		// Remove empty index in buffer by moving next alarms.
		// IF positions in buffer are not empty (trigger false)
		diWarningLoop := diBufferIdToRemove;
		
		WHILE diWarningLoop < HEVS_PackTag_GVL.C_ADMIN_MAXWARNINGS AND 
              stAdminWarning[diWarningLoop + 1].Trigger       DO
			// Cannot be out of buffer because diAlarmLoop < GVL_PackConstant.ALARM_EXTENT
			// Move buffer (n+1) to buffer(n)
			stAdminWarning[diWarningLoop] := stAdminWarning[diWarningLoop + 1]; 
			diWarningLoop := diWarningLoop + 1;
		END_WHILE
		
		// Erase last position on buffer.
		IF diWarningLoop <> diBufferIdToRemove THEN
			stAdminWarning[diWarningLoop].AckDateTime := DT#1970-1-1-0:0:0;
			stAdminWarning[diWarningLoop].Category := 0;
			stAdminWarning[diWarningLoop].DateTime := DT#1970-1-1-0:0:0;
			stAdminWarning[diWarningLoop].ID := 0;
			stAdminWarning[diWarningLoop].Message := '';
			stAdminWarning[diWarningLoop].Trigger := FALSE;
			stAdminWarning[diWarningLoop].Value := 0;
		END_IF
	END_IF 
END_IF

(*
	Set AckDateTime
	Do not set if NOT bSetAlarm because Event was removed with the above code.
	
	Acknowledge on rising edge only
*)
rTrigAck(CLK := bAckWarningTrig);

IF rTrigAck.Q AND bSetWarning THEN
	FOR diWarningLoop := 0 TO HEVS_PackTag_GVL.C_ADMIN_MAXWARNINGS BY 1 DO
		IF (stAdminWarning[diWarningLoop].ID = ID) THEN
			stAdminWarning[diWarningLoop].AckDateTime := PackTag.Admin.PLCDateTime;
		END_IF
	END_FOR	
END_IF


                
END_FUNCTION_BLOCK

(* A function block to set an alarm using PackML 2022 structure TwinCAT Tc3_EventLogger Source: www.hevs.ch Author: Cedric Lenoir Date: 22 August 2024 *)
FUNCTION_BLOCK FB_HEVS_StopReason
  VAR_INPUT
    SuspendCategory : DINT := 1;  (* With default value 1 *)
    HoldCategory : DINT := 2;  (* With default value 2 *)
    StopCategory : DINT := 3;  (* With default value 3 *)
    AbortCategory : DINT := 4;  (* With default value 4 *)
    CompleteCategory : DINT := 6;  (* With default value 6 *)
  END_VAR
  VAR_IN_OUT
    stStopReason : HEVS_PackTag_Event;
    stAdminAlarm : ARRAY[0..HEVS_PackTag_GVL.C_ADMIN_MAXALARMS] OF HEVS_PackTag_Event;
  END_VAR
  VAR_OUTPUT
    SuspendCmd : BOOL;
    HoldCmd : BOOL;
    StopCmd : BOOL;
    AbortCmd : BOOL;
    CompleteCmd : BOOL;
    stopReasonToMaster : E_PackCmd := E_PackCmd.eUndefined;  (* Use to activate Stop Reason on FB_PackMasterState *)
  END_VAR
  VAR
    SuspendExistInAlarm : BOOL;
    HoldExistInAlarm : BOOL;
    StopExistInAlarm : BOOL;
    AbortExistInAlarm : BOOL;
    CompleteExistInAlarm : BOOL;
    SuspendId : DINT;
    HoldId : DINT;
    StopId : DINT;
    AbortId : DINT;
    CompleteId : DINT;
    diAlarmLoop : DINT;
  END_VAR

                  (*
	TR 88 not precise, 
	we will show the Cmd with the Highest Priority
	with Abort, the higest, Stop, Complete, Hold and Suspend, the lowest.
*)
SuspendExistInAlarm := FALSE;
HoldExistInAlarm := FALSE;
StopExistInAlarm := FALSE;
AbortExistInAlarm := FALSE;
CompleteExistInAlarm := FALSE;

SuspendId := 0;
HoldId := 0;
StopId := 0;
AbortId := 0;
CompleteId := 0;
	
FOR diAlarmLoop := 0 TO HEVS_PackTag_GVL.C_ADMIN_MAXALARMS BY 1 DO
	IF stAdminAlarm[diAlarmLoop].Category = SuspendCategory THEN
		SuspendExistInAlarm := TRUE;
		SuspendId := diAlarmLoop;
	END_IF

	IF stAdminAlarm[diAlarmLoop].Category = HoldCategory THEN
		HoldExistInAlarm := TRUE;
		HoldId := diAlarmLoop;
	END_IF

	IF stAdminAlarm[diAlarmLoop].Category = StopCategory THEN
		StopExistInAlarm := TRUE;
		StopId := diAlarmLoop;
	END_IF

	IF stAdminAlarm[diAlarmLoop].Category = AbortCategory THEN
		AbortExistInAlarm := TRUE;
		AbortId := diAlarmLoop;
	END_IF

	IF stAdminAlarm[diAlarmLoop].Category = CompleteCategory THEN
		CompleteExistInAlarm := TRUE;
		CompleteId := diAlarmLoop;
	END_IF
END_FOR

// Select the highest priority sto reason
IF AbortExistInAlarm THEN
	stStopReason := stAdminAlarm[AbortId];
	stopReasonToMaster := E_PackCmd.eAbort;
	
ELSIF StopExistInAlarm THEN
	stStopReason := stAdminAlarm[StopId];
	stopReasonToMaster := E_PackCmd.eStop;

ELSIF CompleteExistInAlarm THEN
	stStopReason := stAdminAlarm[CompleteId];
	stopReasonToMaster := E_PackCmd.eComplete;
	
ELSIF HoldExistInAlarm THEN
	stStopReason := stAdminAlarm[HoldId];
	stopReasonToMaster := E_PackCmd.eHold;
	
ELSIF SuspendExistInAlarm THEN
	stStopReason := stAdminAlarm[SuspendId];
	stopReasonToMaster := E_PackCmd.eSuspend;
	
ELSE // No Stop reason, reset
	stStopReason.AckDateTime := DT#1970-1-1-0:0:0;
	stStopReason.Category := 0;
	stStopReason.DateTime := DT#1970-1-1-0:0:0;
	stStopReason.ID := 0;
	stStopReason.Message := '';
	stStopReason.Trigger := FALSE;
	stStopReason.Value := 0; 

	stopReasonToMaster := E_PackCmd.eUndefined;
END_IF

(*
	Set outputs
*)
AbortCmd := AbortExistInAlarm;
StopCmd := StopExistInAlarm AND NOT AbortExistInAlarm;
CompleteCmd := CompleteExistInAlarm AND NOT (AbortExistInAlarm OR StopExistInAlarm);
HoldCmd := HoldExistInAlarm AND NOT (AbortExistInAlarm OR StopExistInAlarm OR CompleteExistInAlarm);
SuspendCmd := SuspendCmd AND NOT (AbortExistInAlarm OR StopExistInAlarm OR CompleteExistInAlarm OR HoldExistInAlarm);



                
END_FUNCTION_BLOCK

(* A function block of type Enable Source: www.hevs.ch Author: Cedric Lenoir Date: 22 August 2024 *)
FUNCTION_BLOCK FB_InOpBase
  VAR_INPUT
    Enable : BOOL;
  END_VAR
  VAR_OUTPUT
    InOperation : BOOL;
    Error : BOOL;
    ErrorId : WORD;
  END_VAR
  VAR
    eOperationBase : E_InOperationBase;
    errorCondition : BOOL;
  END_VAR

                  // Read Input

CASE eOperationBase OF
	E_InOperationBase.Idle 			:
		IF Enable THEN
			eOperationBase := E_InOperationBase.Init;
		END_IF
        
	E_InOperationBase.Init 			:
		IF NOT Enable THEN
			eOperationBase := E_InOperationBase.Idle;
		ELSIF errorCondition THEN
			eOperationBase := E_InOperationBase.Error;
		END_IF
        
	E_InOperationBase.InOp  :
		IF NOT Enable THEN
			eOperationBase := E_InOperationBase.Idle;
		ELSIF errorCondition THEN
			eOperationBase := E_InOperationBase.Error;
		END_IF
        
	E_InOperationBase.Error			:
		IF NOT Enable THEN
			eOperationBase := E_InOperationBase.Idle;
		END_IF
END_CASE

InOperation := eOperationBase = E_InOperationBase.InOp;
			   
Error := (eOperationBase = E_InOperationBase.Error);

// 0 while no ID defined
ErrorId := 0;
                
END_FUNCTION_BLOCK

PROGRAM PRG_Sandbox
  VAR
    uliLoop : ULINT;
    bInit : BOOL;  (* Only used to give a basic value to some variables. *)
    fbInOpBase : FB_InOpBase;
    fbExecuteDone : FB_ExecuteDone;
  END_VAR

                  (*
    Test base FB
*)
fbInOpBase();
fbExecuteDone();

uliLoop := uliLoop + 1;
(*
    Used to test connection with Node-RED via ADS
*)
ACT_TestNode();


                

ACTION ACT_TestNode:
                      (*
    This part is only used to test the communication with Node-RED
*)
IF NOT bInit THEN
    bInit := TRUE;
    GVL_Node.readREAL    := 3.14;
    GVL_Node.readDINT    := 421;
    GVL_Node.readBOOL    := TRUE;
    GVL_Node.readString  := 'Empty';
    GVL_Node.writeREAL   := 0;
    GVL_Node.writeDINT   := 0;
    GVL_Node.writeBOOL   := FALSE;
END_IF

IF GVL_Node.readREAL > 6.28 THEN
    GVL_Node.readREAL := 0;
ELSE
    GVL_Node.readREAL := GVL_Node.readREAL + 0.1; ;
END_IF
    
IF GVL_Node.readDINT > 1000 THEN
    GVL_Node.readDINT := 0;
ELSE
    GVL_Node.readDINT := GVL_Node.readDINT + 1;
END_IF
                    
END_ACTION
END_PROGRAM

(* www.hevs.ch Institut Systemes Industriels Project: HEVS Pack 2022 Author: Cedric Lenoir Date: 2024 August 29 This program is done to test alarms with a set of 3 Alarms 3 Warnings *)
PROGRAM PRG_TestAlarm
  VAR
    BuildUiString : STRING;  (* Tempo var to display an evant in String Format for UI *)
    fbSetAlarm_0 : FB_HEVS_SetAlarm;  (* Test alarms with FB first *)
    fbSetAlarm_1 : FB_HEVS_SetAlarm;
    fbSetAlarm_2 : FB_HEVS_SetAlarm;
    fbSetWarning_0 : FB_HEVS_SetWarning;
    fbSetWarning_1 : FB_HEVS_SetWarning;
    fbSetWarning_2 : FB_HEVS_SetWarning;
  END_VAR

                  (*
	Call some alarms for test
*) 
fbSetAlarm_0(// Bit activation of Alarm and Ack
			 bSetAlarm := PackTag.hevsPackAlarm_UI.uiSetAlarm_0,
	         bAckAlarmTrig := PackTag.hevsPackAlarm_UI.uiAckAlarm_0,
			 // Alarm Parameters
			 ID := 5,
	         Value := 35,
	         Message := 'Abort 4, E-Stop',
	         Category := E_EventCategory.Abort,
			 // Reference to plc time from PackTag
			 plcDateTimePack	:= PackTag.Admin.PLCDateTime,
			 // Link to PackTag Admin
	         stAdminAlarm := PackTag.Admin.Alarm,
			 stAdminAlarmHistory := PackTag.Admin.AlarmHistory);
			 
fbSetAlarm_1(bSetAlarm := PackTag.hevsPackAlarm_UI.uiSetAlarm_1,
	         bAckAlarmTrig := PackTag.hevsPackAlarm_UI.uiAckAlarm_1,
			 ID := 6,
	         Value := 36,
	         Message := 'Stop 3, Motor Hot',
	         Category := E_EventCategory.Stop,
			 // Reference to plc time from PackTag
			 plcDateTimePack	:= PackTag.Admin.PLCDateTime,
			 // Link to PackTag Admin
	         stAdminAlarm := PackTag.Admin.Alarm,
			 stAdminAlarmHistory := PackTag.Admin.AlarmHistory);


fbSetAlarm_2(bSetAlarm := PackTag.hevsPackAlarm_UI.uiSetAlarm_2,
	         bAckAlarmTrig := PackTag.hevsPackAlarm_UI.uiAckAlarm_2,
			 ID := 7,
	         Value := 37,
	         Message := 'Hold 2, Gripper not closed',
	         Category := E_EventCategory.Hold,
			 // Reference to plc time from PackTag
			 plcDateTimePack	:= PackTag.Admin.PLCDateTime,
			 // Link to PackTag Admin
	         stAdminAlarm := PackTag.Admin.Alarm,
			 stAdminAlarmHistory := PackTag.Admin.AlarmHistory);	

(*
	Call some warnings for test
*)
fbSetWarning_0(bSetWarning := PackTag.hevsPackAlarm_UI.uiSetWarning_0,
	           bAckWarningTrig := PackTag.hevsPackAlarm_UI.uiAckWarning_0,
			   // Warning Parameters
			   ID := 1,
	           Value := 31,
	           Message := 'Warning 0, Door Open',
	           Category := E_EventCategory.Warning,
			   // Reference to plc time from PackTag
			   plcDateTimePack	:= PackTag.Admin.PLCDateTime,
			   // Link to PackTag Admin
	           stAdminWarning := PackTag.Admin.Warning);
			 
fbSetWarning_1(bSetWarning := PackTag.hevsPackAlarm_UI.uiSetWarning_1,
	           bAckWarningTrig := PackTag.hevsPackAlarm_UI.uiAckWarning_1,
			   // Warning Parameters
			   ID := 2,
	           Value := 32,
	           Message := 'Warning 1, Loaded',
	           Category := E_EventCategory.Warning,
			   // Reference to plc time from PackTag
			   plcDateTimePack	:= PackTag.Admin.PLCDateTime,
			   // Link to PackTag Admin
	           stAdminWarning := PackTag.Admin.Warning);


fbSetWarning_2(bSetWarning := PackTag.hevsPackAlarm_UI.uiSetWarning_2,
	           bAckWarningTrig := PackTag.hevsPackAlarm_UI.uiAckWarning_2,
			   // Warning Parameters
			   ID := 3,
	           Value := 33,
	           Message := 'Warning 3, Finished',
	           Category := E_EventCategory.Warning,
			   // Reference to plc time from PackTag
			   plcDateTimePack	:= PackTag.Admin.PLCDateTime,
			   // Link to PackTag Admin
	           stAdminWarning := PackTag.Admin.Warning);						 

// Display first evant in UI in string format.
// Could add History too.
ACT_Build_Ui_Strings();


			 		 

                

ACTION ACT_Build_Ui_Strings:
                      (*
	Send to UI:	First line of Alarms
				First line of Warning
				Stop reason
*)
//PackTag.hevsPackAlarm_UI.uiTextAlarmOne := 'Complete with first Alarm';
BuildUiString := DINT_TO_STRING(PackTag.Admin.Alarm[0].ID);
BuildUiString := CONCAT(BuildUiString, ' ');
BuildUiString := CONCAT(BuildUiString, PackTag.Admin.Alarm[0].Message);
BuildUiString := CONCAT(BuildUiString, ' ');
BuildUiString := CONCAT(BuildUiString, DINT_TO_STRING(PackTag.Admin.Alarm[0].Category));
BuildUiString := CONCAT(BuildUiString, ' ');
BuildUiString := CONCAT(BuildUiString, DT_TO_STRING(PackTag.Admin.Alarm[0].DateTime));
PackTag.hevsPackAlarm_UI.uiTextAlarmOne := BuildUiString; 


BuildUiString := DINT_TO_STRING(PackTag.Admin.Warning[0].ID);
BuildUiString := CONCAT(BuildUiString, ' ');
BuildUiString := CONCAT(BuildUiString, PackTag.Admin.Warning[0].Message);
BuildUiString := CONCAT(BuildUiString, ' ');
BuildUiString := CONCAT(BuildUiString, DINT_TO_STRING(PackTag.Admin.Warning[0].Category));
BuildUiString := CONCAT(BuildUiString, ' ');
BuildUiString := CONCAT(BuildUiString, DT_TO_STRING(PackTag.Admin.Warning[0].DateTime));
PackTag.hevsPackAlarm_UI.uiTextWarningOne := BuildUiString;

BuildUiString := DINT_TO_STRING(PackTag.Admin.StopReason.ID);
BuildUiString := CONCAT(BuildUiString, ' ');
BuildUiString := CONCAT(BuildUiString, PackTag.Admin.StopReason.Message);
BuildUiString := CONCAT(BuildUiString, ' ');
BuildUiString := CONCAT(BuildUiString, DINT_TO_STRING(PackTag.Admin.StopReason.Category));
BuildUiString := CONCAT(BuildUiString, ' ');
BuildUiString := CONCAT(BuildUiString, DT_TO_STRING(PackTag.Admin.StopReason.DateTime));
PackTag.hevsPackAlarm_UI.uiTextStopReason := BuildUiString;


                    
END_ACTION
END_PROGRAM

(* www.hevs.ch Institut Systemes Industriels Project: HEVS Pack 2022 Author: Cedric Lenoir Date: 2024 August 30 This Function Block compute time statistics *)
FUNCTION_BLOCK FB_PackStatistic
  VAR_INPUT
    Enable : BOOL;
  END_VAR
  VAR_IN_OUT
    plcCurrentTime_s : UDINT;  (* E.g from PackTag.hevsPackTime.Local_date_time_seconds *)
    unitCurrentMode : E_PackModes;
    unitCurrentState : E_PackState;
    unitAdmin : HEVS_PackTag_Admin;
  END_VAR
  VAR_OUTPUT
    Active : BOOL;
  END_VAR
  VAR
    trigModeTimeCurrent : R_TRIG;  (* Detext State / Mode change *)
    trigStateTimeCurrent : R_TRIG;
    memCurrentMode : E_PackModes := E_PackModes.Invalid;
    memCurrentState : E_PackState := E_PackState.eUndefined;
    timeModeAtTrigger_s : UDINT;  (* Start time at trigger to compute current *)
    timeStateAtTrigger_s : UDINT;
    bProgramStarted : BOOL;
    timeProgramStarted_s : UDINT;
    getMemCumTimeMode : DINT;  (* Get Time In CumulativeTime for Mode and or state *)
    getMemCumTimeModeState : DINT;
  END_VAR

                  IF Enable THEN
	trigModeTimeCurrent(clk := (unitCurrentMode <> memCurrentMode));
	trigStateTimeCurrent(clk := (unitCurrentState <> memCurrentState));
	
	IF trigModeTimeCurrent.Q THEN
		timeModeAtTrigger_s := plcCurrentTime_s;
		memCurrentMode := unitCurrentMode;
		// Get Stored value to compute new cummulative time.
		getMemCumTimeMode := unitAdmin.CumulativeTime[0].ModeStateTimes[unitCurrentMode].Mode;
	END_IF
	
	IF trigStateTimeCurrent.Q THEN
		timeStateAtTrigger_s := plcCurrentTime_s;
		memCurrentState := unitCurrentState;
	END_IF
	
	// If mode or state changed
	IF trigModeTimeCurrent.Q  OR
	   trigStateTimeCurrent.Q THEN
	   getMemCumTimeModeState := unitAdmin.CumulativeTime[0].ModeStateTimes[unitCurrentMode].State[memCurrentState];
	END_IF
	
	IF NOT bProgramStarted THEN
		bProgramStarted := TRUE;
		timeProgramStarted_s := plcCurrentTime_s;
	END_IF
	
	unitAdmin.ModeTimeCurrent := UDINT_TO_DINT(plcCurrentTime_s - timeModeAtTrigger_s);
	
	unitAdmin.StateTimeCurrent := UDINT_TO_DINT(plcCurrentTime_s - timeStateAtTrigger_s);
	
	// Default for [*] time from start program
	// No retain, that is number of Sec since last restart.
	unitAdmin.CumulativeTime[0].AccTimeSinceReset := UDINT_TO_DINT(plcCurrentTime_s - timeProgramStarted_s);
	
	// Minimum protection in case of unitCurrentMode exceed 
	//	HEVS_PackTag_GVL.C_MAXMODSTATESTIMES
	IF unitCurrentMode <= HEVS_PackTag_GVL.C_MAXMODSTATESTIMES THEN
		// getMemCumTimeMode is set only at trigger change mode
		unitAdmin.CumulativeTime[0].ModeStateTimes[unitCurrentMode].Mode := getMemCumTimeMode + unitAdmin.ModeTimeCurrent;
	END_IF
	
	// Minimum protection in case of unitCurrentMode exceed 
	//	HEVS_PackTag_GVL.C_MAXMODSTATESTIMES
	// 	HEVS_PackTag_GVL.C_MAXSTATES
	IF unitCurrentMode <= HEVS_PackTag_GVL.C_MAXMODSTATESTIMES AND
	   unitCurrentState <= HEVS_PackTag_GVL.C_MAXSTATES        THEN
		// getMemCumTimeModeState is set only at trigger change of mode OR state 
		unitAdmin.CumulativeTime[0].ModeStateTimes[unitCurrentMode].State[unitCurrentState] := getMemCumTimeModeState +  unitAdmin.StateTimeCurrent;
	END_IF
	
	Active	:= FALSE;
ELSE
	
	Active	:= TRUE;
END_IF




                
END_FUNCTION_BLOCK

(* www.hevs.ch Institut Systemes Industriels Project: HEVS Pack 2022 Author: Cedric Lenoir Date: 2024 August 06 Summary: Used to test and simulate first version of PackMaster Does nothing in Waitstates Wait 2.5 secoond before to return SC in *)
FUNCTION_BLOCK FB_ModuleAxis
  VAR_INPUT
    resetSafePosition : LREAL;
    absolutePosition : LREAL;
    absolutePickStart : BOOL;
    stSetParam : ST_SetMotionParam;
  END_VAR
  VAR_IN_OUT
    axisRef : MB_AXISIF_REF;
    Status_StateCurrent : DINT;  (* has to take the PackTag Status.StateCurrent *)
    Status_ModeCurrent : DINT;
  END_VAR
  VAR_OUTPUT
    absPositionDone : BOOL;
    absIsPosition : LREAL;  (* Return actual position of the axis *)
  END_VAR
  VAR
    stateLastCycie : E_PackState := E_PackState.eUndefined;  (* Store last cycle at the en of FB call to detect and state change Used to force minimum of one testSC.In = 0 and reset SC once between each SC *)
    actualState : E_PackState := E_PackState.eAborted;
    actualMode : E_PackModes := E_PackModes.Production;
    init : BOOL;
    testSC : TON;
    setSC : BOOL;  (* This Flag is used as result on SC State complete. *)
    stActing : ST_Acting;
    mcReadActualPos : MC_ReadActualPosition;  (* List of Function Blocks *)
    mcReadStatus : MC_ReadStatus;
    mcPower : MC_Power;
    mcMoveAbs : MC_MoveAbsolute;
    mcStop : MC_Stop := (Deceleration := 1);
    mcReset : MC_Reset;
    axisAborting : E_AxisAborting;  (* List of enum for internal states of axes *)
    axisClearing : E_AxisClearing;
    axisResetting : E_AxisResetting;  (* Go to safe position *)
    axisStarting : E_AxisStarting;  (* Go to firs corner *)
    axisStopping : E_AxisStopping;
    axisExecute : E_AxisExecute;
    calibrationCounter : DINT;  (* For motion calibration *)
    calibrationIncrement : REAL;
  END_VAR

                  IF NOT init THEN
    init := TRUE;
END_IF

actualState := Status_StateCurrent;
actualMode := Status_ModeCurrent;

// State machine is implicit because transitions are not set by this FB
// That is: a CASE OF does not have place here

// Eacn State is called via and ACTion with 
//	Condition of state
//	Reset of internal state machine when not used
//	That's why, ACTion MUST not be called in a CASE..OF
//  Order of ACTion is not important, because only one should be executed 
//  In any state
// 
//	IF actualState = E_PackState.eUnsuspending THEN
	// Set to TRUE if no action requested
//	stActing.Unsuspending_SC := TRUE;
//	END_IF

ACT_Aborting();
ACT_Clearing();
ACT_Completing();
ACT_Execute();
ACT_Holding();
ACT_Resetting();
ACT_Starting();
ACT_Stopping();
ACT_Suspending();
ACT_Unholding();
ACT_Unsuspending();

(**********************************************************************************************************************
	Axis
**********************************************************************************************************************)
mcReadStatus(Axis := axisRef,
		     Enable := TRUE);

mcReadActualPos(Axis := axisRef,
                Enable := TRUE,
                Position => absIsPosition);

mcPower(Axis := axisRef,
		Enable := NOT (actualState = E_PackState.eAborted) 		  AND
 				  // In aborting, do not disable while stopping
				  NOT ((actualState = E_PackState.eAborting) AND
                       NOT (axisAborting = E_AxisAborting.eStopping)) AND
				  // E_AxisClearing.eErrorStop should be possible
				  // if actualState = E_PackState.eClearing
				  NOT (axisClearing = E_AxisClearing.eErrorStop));

mcStop(Axis := axisRef,
	   // Stop in case of Stopping
	   // Stop in case of Aborting (before to Disable
	   Deceleration := stSetParam.rDeceleration_m_s2,	   		
       Execute := (axisStopping = E_AxisStopping.eStopping) OR
                  (axisAborting = E_AxisAborting.eStopping));

mcReset(Axis := axisRef,
        Execute := (axisClearing = E_AxisClearing.eErrorStop) OR
                    axisAborting = E_AxisAborting.eErrorStop);

mcMoveAbs(Axis := axisRef,
          Velocity := stSetParam.rVelocity_m_s,
          Acceleration := stSetParam.rAcceleration_m_s2,
          Deceleration := stSetParam.rDeceleration_m_s2,
          Jerk := stSetParam.rJerk_m_s3); 
		  
mcMoveAbs.Execute := (axisExecute = E_AxisExecute.eSetAbsolutePosition) OR
					 (axisResetting = E_AxisResetting.eMotionInit) 		OR
					 (axisStarting = E_AxisStarting.eMotionStarting)    OR
					 absolutePickStart;
(*
	Manage State Complete at the end of the Function Block
*)
			
// For test of State Machine, we use a timer.
// Its allow to have some time to visualise it
// We should remove this timer in production version
testSC(IN := stActing.Clearing_SC 		OR
             stActing.Starting_SC      	OR
             stActing.Execute_SC       	OR
             stActing.Stopping_SC      	OR
             stActing.Aborting_SC      	OR
             stActing.Holding_SC       	OR
             stActing.Unholding_SC     	OR
             stActing.Suspending_SC		OR
             stActing.Unsuspending_SC	OR
             stActing.Resetting_SC     	OR
             stActing.Completing_SC,
        PT := T#2500MS); 

// State Complete if setSC is TRUE,
setSC := testSC.Q AND (stateLastCycie = actualState);

// This Statement MUST be written AFTER evaluation of setSC
stateLastCycie := actualState;



                

ACTION ACT_Clearing:
                      (*
	Manage Clearing
*)

// actualState is actual state of Unit from:
//	PackTag.Status.StateCurrent
//
// Wait for : stActing.Clearing_SC : TRUE
// While not all units SC, actualState remains in eClearing.
//
// From PLCopen Motion, the axis at start could be
// Standstill	--> Enabled
// Disabled		--> Need an enable for SC
// ErrorStop	--> Need a reset befoire to be enabled
IF actualState = E_PackState.eClearing THEN
	CASE axisClearing OF
		E_AxisClearing.eIdle :
			IF mcReadStatus.Standstill THEN
				axisClearing := E_AxisClearing.eEnabled;
			ELSIF mcReadStatus.ErrorStop THEN
				axisClearing := E_AxisClearing.eErrorStop;
			ELSE
				axisClearing := E_AxisClearing.eDisabled;
			END_IF
		
		E_AxisClearing.eErrorStop :
			IF mcReadStatus.Standstill THEN
				axisClearing := E_AxisClearing.eEnabled;
			ELSE
				axisClearing := E_AxisClearing.eDisabled;
			END_IF
		
		E_AxisClearing.eDisabled  :
			IF mcReadStatus.Standstill THEN
				axisClearing := E_AxisClearing.eEnabled;
			ELSIF mcReadStatus.ErrorStop THEN
				axisClearing := E_AxisClearing.eErrorStop;
			END_IF
		
		E_AxisClearing.eEnabled   :
			IF mcReadStatus.ErrorStop THEN
				axisClearing := E_AxisClearing.eErrorStop;
			END_IF
	END_CASE
	stActing.Clearing_SC := (axisClearing = E_AxisClearing.eEnabled);
ELSE
	stActing.Clearing_SC := FALSE;
	axisClearing := E_AxisClearing.eIdle; 
END_IF

                    
END_ACTION

ACTION ACT_Starting:
                      (*
	Manage Starting
*)
IF actualState = E_PackState.eStarting THEN
	CASE axisStarting OF
		E_AxisStarting.eIdle :
			axisStarting := E_AxisStarting.eMotionStarting;
			
		E_AxisStarting.eMotionStarting :
			IF mcMoveAbs.Done THEN
				axisStarting := E_AxisStarting.eMotionStartingDone;
			END_IF;
	
		E_AxisStarting.eMotionStartingDone :
			;
	
	END_CASE
	stActing.Starting_SC := (axisStarting = E_AxisStarting.eMotionStartingDone);
ELSE
	stActing.Starting_SC := FALSE;
	axisStarting := E_AxisStarting.eIdle;
END_IF
                    
END_ACTION

ACTION ACT_Execute:
                      (*
	Manage Execute
*)
IF (actualState = E_PackState.eExecute)  AND
   (actualMode = E_PackModes.Manual)     THEN
	CASE axisExecute OF
		E_AxisExecute.eIdle :
			axisExecute := E_AxisExecute.eSetAbsolutePosition;
			mcMoveAbs.Position := absolutePosition;
			
		E_AxisExecute.eSetAbsolutePosition :
			IF mcMoveAbs.Done THEN
				axisExecute := E_AxisExecute.eSetAbsolutePositionDone;
			END_IF;
	
		E_AxisExecute.eSetAbsolutePositionDone :
			axisExecute := E_AxisExecute.eIdle;

	END_CASE
	absPositionDone := axisExecute = E_AxisExecute.eSetAbsolutePositionDone;
ELSE
	axisExecute := E_AxisExecute.eIdle;
END_IF

IF (actualState = E_PackState.eExecute)  AND
   (actualMode = E_PackModes.Production) THEN
    mcMoveAbs.Position := absolutePosition;
	absPositionDone := mcMoveAbs.Done                                      AND 
                       (mcReadActualPos.Position - 0.1 < absolutePosition) AND
                       (mcReadActualPos.Position + 0.1 > absolutePosition);
END_IF
                    
END_ACTION

ACTION ACT_Stopping:
                      (*
	Manage Stopping
*)
IF actualState = E_PackState.eStopping THEN
	CASE axisStopping OF
		E_AxisStopping.eIdle :
			IF mcReadStatus.Disabled THEN
				axisStopping := E_AxisStopping.eStopped;
			ELSIF mcReadStatus.ErrorStop THEN
				axisStopping := E_AxisStopping.eStopped;
			ELSIF mcReadStatus.Standstill THEN
				axisStopping := E_AxisStopping.eStopped;
			ELSE 
				axisStopping := E_AxisStopping.eStopping;
			END_IF
		E_AxisStopping.eStopping :
			IF mcReadStatus.Disabled THEN
				axisStopping := E_AxisStopping.eStopped;
			ELSIF mcReadStatus.ErrorStop THEN
				axisStopping := E_AxisStopping.eStopped;
			ELSIF mcReadStatus.Standstill THEN
				axisStopping := E_AxisStopping.eStopped;
			END_IF;
	
		E_AxisStopping.eStopped :
			;
	
	END_CASE
	stActing.Stopping_SC := (axisStopping = E_AxisStopping.eStopped);
ELSE
	stActing.Stopping_SC := FALSE;
	axisStopping := E_AxisStopping.eIdle;
END_IF
                    
END_ACTION

ACTION ACT_Aborting:
                      (*
	Manage Aborting
*)
IF actualState = E_PackState.eAborting THEN
	CASE axisAborting OF
		E_AxisAborting.eIdle :
			IF mcReadStatus.Disabled THEN
				axisAborting := E_AxisAborting.eDisabled;
			ELSIF mcReadStatus.ErrorStop THEN
				axisAborting := E_AxisAborting.eErrorStop;
			ELSIF mcReadStatus.Standstill THEN
				axisAborting := E_AxisAborting.eStandstill;
			ELSE 
				axisAborting := E_AxisAborting.eStopping;
			END_IF
		E_AxisAborting.eStopping :
			IF mcReadStatus.Disabled THEN
				axisAborting := E_AxisAborting.eDisabled;
			ELSIF mcReadStatus.ErrorStop THEN
				axisAborting := E_AxisAborting.eErrorStop;
			ELSIF mcReadStatus.Standstill THEN
				axisAborting := E_AxisAborting.eStandstill;
			END_IF;
	
		E_AxisAborting.eStandstill :
			IF mcReadStatus.Disabled THEN
				axisAborting := E_AxisAborting.eDisabled;
			ELSIF mcReadStatus.ErrorStop THEN
				axisAborting := E_AxisAborting.eErrorStop;
			END_IF;;
	
		E_AxisAborting.eErrorStop :
			IF mcReadStatus.Disabled THEN
				axisAborting := E_AxisAborting.eDisabled;
			ELSIF mcReadStatus.Standstill THEN
				axisAborting := E_AxisAborting.eStandstill;
			END_IF;;
	
		E_AxisAborting.eDisabled :
//			IF mcReadStatus.ErrorStop THEN
//				axisAborting := E_AxisAborting.eErrorStop;
//			END_IF		
			;
	END_CASE
	stActing.Aborting_SC := (axisAborting = E_AxisAborting.eDisabled);
ELSE
	stActing.Aborting_SC := FALSE;
	axisAborting := E_AxisAborting.eIdle;
END_IF

                    
END_ACTION

ACTION ACT_Holding:
                      (*
	Manage Holding
*)
IF actualState = E_PackState.eHolding THEN
	// Set to TRUE if no action requested
	stActing.Holding_SC := TRUE;
ELSE
	stActing.Holding_SC := FALSE;
END_IF

                    
END_ACTION

ACTION ACT_Unholding:
                      (*
	Manage Unholding
*)
IF actualState = E_PackState.eUnholding THEN
	// Set to TRUE if no action requested
	stActing.Unholding_SC := TRUE;
END_IF

                    
END_ACTION

ACTION ACT_Suspending:
                      (*
	Manage Suspending
*)
IF actualState = E_PackState.eSuspending THEN
	// Set to TRUE if no action requested
	stActing.Suspending_SC := TRUE;
END_IF
                    
END_ACTION

ACTION ACT_Unsuspending:
                      (*
	Manage Unsuspending
*)
IF actualState = E_PackState.eUnsuspending THEN
	// Set to TRUE if no action requested
	stActing.Unsuspending_SC := TRUE;
END_IF

                    
END_ACTION

ACTION ACT_Resetting:
                      (*
	Manage Resetting
*)
IF actualState = E_PackState.eResetting THEN
	CASE axisResetting OF
		E_AxisResetting.eIdle :
		    mcMoveAbs.Position := resetSafePosition;
			axisResetting := E_AxisResetting.eMotionInit;
			
		E_AxisResetting.eMotionInit :
			IF mcMoveAbs.Done THEN
				axisResetting := E_AxisResetting.eMotionInitDone;
			END_IF;
	
		E_AxisResetting.eMotionInitDone :
			;
	
	END_CASE
	stActing.Resetting_SC := (axisResetting = E_AxisResetting.eMotionInitDone);
ELSE
	stActing.Resetting_SC := FALSE;
	axisResetting := E_AxisResetting.eIdle;
END_IF
                    
END_ACTION

ACTION ACT_Completing:
                      (*
	Manage Completing
*)
IF actualState = E_PackState.eCompleting THEN
	// Set to TRUE if no action requested
	stActing.Completing_SC := TRUE;
END_IF

                    
END_ACTION

PROPERTY SC : BOOL
GET
                          SC := setSC;
                        
END_GET
END_PROPERTY
END_FUNCTION_BLOCK

(* www.hevs.ch Institut Systemes Industriels Project: Projet No: PW Move Absolute Author: Cedric Lenoir Date: 2024 April 02 Summary: Template of a program using PLCopen on partial Pack State Use a Cyclic Setpoint for motion in Pack Execute. *)
PROGRAM PRG_Process
  VAR
    bStartAbsolutePosition : BOOL;  (* ********************************************************************************************************************* YOUR VARIABLES HERE ********************************************************************************************************************* *)
    bIdle : BOOL;
    stSetParam : ST_SetMotionParam := (rVelocity_m_s := 0.2, rAcceleration_m_s2 := 0.5, rDeceleration_m_s2 := 0.5, rJerk_m_s3 := 1);
    idInList_XYZ : UINT := 1;  (* Nest positions *)
    up_Z_Position : LREAL := -10;
    nestNumber : UINT := 5;
    arListXYZ_Offset : ARRAY[0..10] OF ST_XYZ_Offset;
    timerGripperOpenClose : TON;
    lrMoveAbs_X : LREAL := 0;  (* Values from User Interface *)
    lrMoveAbs_Y : LREAL := 0;
    lrMoveAbs_Z : LREAL := 100;
    eManualJog : E_ManualJog;
    eUnitMove : E_UnitMoveForPickAndPlace := E_UnitMoveForPickAndPlace.Idle;
    uliCount : ULINT;
    bInitDone : BOOL;
    fbModuleAxis_X : FB_ModuleAxis;  (* Pack Partial state machine *)
    fbModuleAxis_Y : FB_ModuleAxis;
    fbModuleAxis_Z : FB_ModuleAxis;
    testMyReal_1 : REAL;
    testMyReal_2 : REAL;
    xOneStep : BOOL;  (* for debug *)
    xEnableStepByStep : BOOL;
    xDisableStepByStop : BOOL;
    xStepByStepMode : BOOL;
    xNextStepEnable : BOOL;
    rTrigNextStep : R_TRIG;
    uliStepCounter : ULINT;
  END_VAR
  VAR CONSTANT
    C_X_StartingPosition : LREAL := -199;
    C_Y_StartingPosition : LREAL := -78;
    C_Z_StartingPosition : LREAL := 0;
    C_Gripper_Open : BOOL := TRUE;
    C_Gripper_Close : BOOL := FALSE;
  END_VAR

                  (* For test only *)
IF NOT bInitDone THEN
	bInitDone := TRUE;
	ACT_InitListOfOffset();
END_IF
testMyReal_2 := testMyReal_1;

(*
	Clearing
	Reset lrMoveAbs_Z lrMoveAbs_Y and lrMoveAbs_X
*)
IF PackTag.Status.StateCurrent = E_PackState.eClearing THEN
	lrMoveAbs_X := C_X_StartingPosition;
	lrMoveAbs_Y := C_Y_StartingPosition;
	lrMoveAbs_Z := C_Z_StartingPosition;
	
	GVL_Abox.uaAboxInterface.uaSchunkGripper.SetOut := TRUE;
END_IF

ACT_OneUnitPick();
ACT_ManualJog();

fbModuleAxis_X(axisRef := GVL_AxisDefines.X_Axis,
			  // Keep actual position of X while resetting.
			  resetSafePosition := fbModuleAxis_X.absIsPosition,
			  // absolutePosition				: LREAL;
			  absolutePickStart := eUnitMove = E_UnitMoveForPickAndPlace.MovePickUpOpen 	OR
								   eUnitMove = E_UnitMoveForPickAndPlace.MoveDownPick 		OR
								   eUnitMove = E_UnitMoveForPickAndPlace.MoveUpPickClosed 	OR
								   eUnitMove = E_UnitMoveForPickAndPlace.MovePlaceUpClosed	OR
								   eUnitMove = E_UnitMoveForPickAndPlace.MoveDownPlace 		OR
								   eUnitMove = E_UnitMoveForPickAndPlace.MoveUpPlace,
			  stSetParam := stSetParam,
			  Status_ModeCurrent := PackTag.Status.UnitModeCurrent,
			  Status_StateCurrent := PackTag.Status.StateCurrent);
			  
fbModuleAxis_Y(axisRef := GVL_AxisDefines.Y_Axis,
			  // Keep actual position of X while resetting.
			  resetSafePosition := fbModuleAxis_Y.absIsPosition,
			  // absolutePosition				: LREAL;
			  absolutePickStart := eUnitMove = E_UnitMoveForPickAndPlace.MovePickUpOpen 	OR
								   eUnitMove = E_UnitMoveForPickAndPlace.MoveDownPick 		OR
								   eUnitMove = E_UnitMoveForPickAndPlace.MoveUpPickClosed 	OR
								   eUnitMove = E_UnitMoveForPickAndPlace.MovePlaceUpClosed	OR
								   eUnitMove = E_UnitMoveForPickAndPlace.MoveDownPlace 		OR
								   eUnitMove = E_UnitMoveForPickAndPlace.MoveUpPlace,
			  stSetParam := stSetParam,
			  Status_ModeCurrent := PackTag.Status.UnitModeCurrent,
			  Status_StateCurrent := PackTag.Status.StateCurrent);

fbModuleAxis_Z(axisRef := GVL_AxisDefines.Z_Axis,
			  resetSafePosition := 100,
			  // absolutePosition				: LREAL;
			  absolutePickStart := eUnitMove = E_UnitMoveForPickAndPlace.MovePickUpOpen 	OR
								   eUnitMove = E_UnitMoveForPickAndPlace.MoveDownPick 		OR
								   eUnitMove = E_UnitMoveForPickAndPlace.MoveUpPickClosed 	OR
								   eUnitMove = E_UnitMoveForPickAndPlace.MovePlaceUpClosed	OR
								   eUnitMove = E_UnitMoveForPickAndPlace.MoveDownPlace 		OR
								   eUnitMove = E_UnitMoveForPickAndPlace.MoveUpPlace,
			  stSetParam := stSetParam,			  
			  Status_ModeCurrent := PackTag.Status.UnitModeCurrent,
			  Status_StateCurrent := PackTag.Status.StateCurrent);

PRG_PackModule_Template(Status_StateCurrent := PackTag.Status.StateCurrent);			  
                

ACTION ACT_OneUnitPick:
                      (*
	Execute Sequence
*)
timerGripperOpenClose(in := (eUnitMove = E_UnitMoveForPickAndPlace.CloseGripper)     OR
	                        (eUnitMove = E_UnitMoveForPickAndPlace.OpenGripperPlace),
					  PT := T#1000MS);


IF xEnableStepByStep THEN
	xEnableStepByStep := FALSE;
	xStepByStepMode := TRUE;
END_IF
IF xDisableStepByStop THEN
	xDisableStepByStop := FALSE;
	xStepByStepMode := FALSE;
END_IF
	
rTrigNextStep(CLk := xOneStep);
IF NOT xStepByStepMode THEN
	xNextStepEnable := TRUE;
ELSE
	xNextStepEnable := rTrigNextStep.Q;
END_IF
IF rTrigNextStep.Q THEN
	xOneStep := FALSE;
	uliStepCounter := uliStepCounter + 1;
END_IF 					  

IF (PackTag.Status.StateCurrent = E_PackState.eExecute)      AND
   (PackTag.Status.UnitModeCurrent = E_PackModes.Production) THEN
	CASE eUnitMove OF
		  E_UnitMoveForPickAndPlace.Idle:
			(* Code for Idle state *)
			IF xNextStepEnable THEN
				eUnitMove := E_UnitMoveForPickAndPlace.InitMove;
			END_IF
			
		  E_UnitMoveForPickAndPlace.InitMove:
			fbModuleAxis_X.absolutePosition := C_X_StartingPosition + arListXYZ_Offset[idInList_XYZ].X_AxisOffsetPosition;
			fbModuleAxis_Y.absolutePosition := C_Y_StartingPosition + arListXYZ_Offset[idInList_XYZ].Y_AxisOffsetPosition;
			fbModuleAxis_Z.absolutePosition := C_Z_StartingPosition + up_Z_Position;
			GVL_Abox.uaAboxInterface.uaSchunkGripper.SetOut := C_Gripper_Open;

			IF xNextStepEnable THEN
				eUnitMove := E_UnitMoveForPickAndPlace.MovePickUpOpen;
			END_IF
 
		  E_UnitMoveForPickAndPlace.MovePickUpOpen:
			(* Code for MovePickUpOpen state *)
			IF fbModuleAxis_X.absPositionDone AND
			   fbModuleAxis_Y.absPositionDone AND
			   fbModuleAxis_Z.absPositionDone AND
			   xNextStepEnable                THEN
			    GVL_Abox.uaAboxInterface.uaSchunkGripper.SetOut := C_Gripper_Open;
				eUnitMove := E_UnitMoveForPickAndPlace.IsUpPickOpen;
			END_IF

		  E_UnitMoveForPickAndPlace.IsUpPickOpen:
			(* Code for IsUpPickOpen state *)
			fbModuleAxis_X.absolutePosition := C_X_StartingPosition + arListXYZ_Offset[idInList_XYZ].X_AxisOffsetPosition;
			fbModuleAxis_Y.absolutePosition := C_Y_StartingPosition + arListXYZ_Offset[idInList_XYZ].Y_AxisOffsetPosition;
			fbModuleAxis_Z.absolutePosition := C_Z_StartingPosition + arListXYZ_Offset[idInList_XYZ].Z_AxisOffsetPosition;

			IF xNextStepEnable THEN
				eUnitMove := E_UnitMoveForPickAndPlace.MoveDownPick;
			END_IF			

		  E_UnitMoveForPickAndPlace.MoveDownPick:
			(* Code for MoveDownPick state *)
			IF fbModuleAxis_X.absPositionDone AND
			   fbModuleAxis_Y.absPositionDone AND
			   fbModuleAxis_Z.absPositionDone AND
			   xNextStepEnable                THEN
				eUnitMove := E_UnitMoveForPickAndPlace.CloseGripper;
			END_IF			

		  E_UnitMoveForPickAndPlace.CloseGripper:
			(* Code for CloseGripper state *)
			GVL_Abox.uaAboxInterface.uaSchunkGripper.SetOut := C_Gripper_Close;
			IF timerGripperOpenClose.Q THEN
				eUnitMove := E_UnitMoveForPickAndPlace.IsClosed;
			END_IF			

		  E_UnitMoveForPickAndPlace.IsClosed:
			(* Code for IsClosed state *)
			fbModuleAxis_X.absolutePosition := C_X_StartingPosition + arListXYZ_Offset[idInList_XYZ].X_AxisOffsetPosition;
			fbModuleAxis_Y.absolutePosition := C_Y_StartingPosition + arListXYZ_Offset[idInList_XYZ].Y_AxisOffsetPosition;
			fbModuleAxis_Z.absolutePosition := C_Z_StartingPosition + up_Z_Position;
			
			IF xNextStepEnable THEN
				eUnitMove := E_UnitMoveForPickAndPlace.MoveUpPickClosed;
			END_IF

		  E_UnitMoveForPickAndPlace.MoveUpPickClosed:
			(* Code for MoveUpPickClosed state *)
			IF fbModuleAxis_X.absPositionDone AND
			   fbModuleAxis_Y.absPositionDone AND
			   fbModuleAxis_Z.absPositionDone AND
			   xNextStepEnable				  THEN
				eUnitMove := E_UnitMoveForPickAndPlace.IsUpPickClosed;
					// Next next here for IsUpPickClosed
					IF idInList_XYZ < nestNumber THEN
						idInList_XYZ := idInList_XYZ + 1;
					ELSE
						idInList_XYZ := 1;
					END_IF
			END_IF				

		  E_UnitMoveForPickAndPlace.IsUpPickClosed:
			(* Code for IsUpPickClosed state *)
			fbModuleAxis_X.absolutePosition := C_X_StartingPosition + arListXYZ_Offset[idInList_XYZ].X_AxisOffsetPosition;
			fbModuleAxis_Y.absolutePosition := C_Y_StartingPosition + arListXYZ_Offset[idInList_XYZ].Y_AxisOffsetPosition;
			fbModuleAxis_Z.absolutePosition := C_Z_StartingPosition + up_Z_Position;

			IF xNextStepEnable THEN
				eUnitMove := E_UnitMoveForPickAndPlace.MovePlaceUpClosed;
			END_IF;				

		  E_UnitMoveForPickAndPlace.MovePlaceUpClosed:
			(* Code for MovePlaceUpClosed state *)
			IF fbModuleAxis_X.absPositionDone AND
			   fbModuleAxis_Y.absPositionDone AND
			   fbModuleAxis_Z.absPositionDone AND 
               xNextStepEnable                THEN
				eUnitMove := E_UnitMoveForPickAndPlace.IsPlaceUpClosed;
			END_IF				

		  E_UnitMoveForPickAndPlace.IsPlaceUpClosed:
			(* Code for IsPlaceUpClosed state *)
			fbModuleAxis_X.absolutePosition := C_X_StartingPosition + arListXYZ_Offset[idInList_XYZ].X_AxisOffsetPosition;
			fbModuleAxis_Y.absolutePosition := C_Y_StartingPosition + arListXYZ_Offset[idInList_XYZ].Y_AxisOffsetPosition;
			fbModuleAxis_Z.absolutePosition := C_Z_StartingPosition + arListXYZ_Offset[idInList_XYZ].Z_AxisOffsetPosition;

			IF xNextStepEnable THEN
				eUnitMove := E_UnitMoveForPickAndPlace.MoveDownPlace;
			END_IF;					

		  E_UnitMoveForPickAndPlace.MoveDownPlace:
			(* Code for MoveDownPlace state *)
			IF fbModuleAxis_X.absPositionDone AND
			   fbModuleAxis_Y.absPositionDone AND
			   fbModuleAxis_Z.absPositionDone AND 
			   xNextStepEnable 				  THEN
				eUnitMove := E_UnitMoveForPickAndPlace.IsMoveDownPlace;
			END_IF			

		  E_UnitMoveForPickAndPlace.IsMoveDownPlace:
			(* Code for IsMoveDownPlace state *)
			GVL_Abox.uaAboxInterface.uaSchunkGripper.SetOut := C_Gripper_Open;
			
			IF xNextStepEnable THEN
				eUnitMove := E_UnitMoveForPickAndPlace.OpenGripperPlace;
			END_IF

		  E_UnitMoveForPickAndPlace.OpenGripperPlace:
			(* Code for OpenGripperPlace state *)
			IF timerGripperOpenClose.Q THEN
				eUnitMove := E_UnitMoveForPickAndPlace.IsOpenGripperPlace;
			END_IF			

		  E_UnitMoveForPickAndPlace.IsOpenGripperPlace:
			(* Code for IsOpenGripperPlace state *)
			fbModuleAxis_X.absolutePosition := C_X_StartingPosition + arListXYZ_Offset[idInList_XYZ].X_AxisOffsetPosition;
			fbModuleAxis_Y.absolutePosition := C_Y_StartingPosition + arListXYZ_Offset[idInList_XYZ].Y_AxisOffsetPosition;
			fbModuleAxis_Z.absolutePosition := C_Z_StartingPosition + up_Z_Position;

			IF xNextStepEnable THEN
				eUnitMove := E_UnitMoveForPickAndPlace.MoveUpPlace;
			END_IF			

		  E_UnitMoveForPickAndPlace.MoveUpPlace:
			(* Code for MoveUpPlace state *)
			IF fbModuleAxis_X.absPositionDone AND
			   fbModuleAxis_Y.absPositionDone AND
			   fbModuleAxis_Z.absPositionDone AND 
               xNextStepEnable                THEN
				eUnitMove := E_UnitMoveForPickAndPlace.IsMoveUpPlace;
			END_IF			

		  E_UnitMoveForPickAndPlace.IsMoveUpPlace:
			(* Code for IsMoveUpPlace state *)
			IF xNextStepEnable THEN
				eUnitMove := E_UnitMoveForPickAndPlace.Idle;
			END_IF

		  E_UnitMoveForPickAndPlace.MotionError:
			(* Code for MotionError state *)
	END_CASE
ELSE
	eUnitMove := E_UnitMoveForPickAndPlace.Idle;
END_IF
                    
END_ACTION

ACTION ACT_ManualJog:
                      (*
	Execute Manual Sequence
*)
IF PackTag.Status.StateCurrent = E_PackState.eExecute 	 AND
   (PackTag.Status.UnitModeCurrent = E_PackModes.Manual) THEN
	CASE eManualJog OF
	E_ManualJog.eIdle :
		IF PackTag.Status.UnitModeCurrent = E_PackModes.Manual THEN
			eManualJog := E_ManualJog.eNextMove;
		END_IF
		
	E_ManualJog.eNextMove :
		fbModuleAxis_Z.absolutePosition := lrMoveAbs_Z;
		eManualJog := E_ManualJog.eMove_Z;
		
	E_ManualJog.eMove_Z :
		IF fbModuleAxis_Z.absPositionDone THEN
			bStartAbsolutePosition := FALSE;
			eManualJog := E_ManualJog.eMove_Z_Done;
		END_IF
		
	E_ManualJog.eMove_Z_Done :;
		fbModuleAxis_X.absolutePosition := lrMoveAbs_X;
		eManualJog := E_ManualJog.eMove_X;
		
	E_ManualJog.eMove_X :;
		IF fbModuleAxis_X.absPositionDone THEN
			eManualJog := E_ManualJog.eMove_X_Done;
		END_IF
		
	E_ManualJog.eMove_X_Done :;
		fbModuleAxis_Y.absolutePosition := lrMoveAbs_Y;
		eManualJog := E_ManualJog.eMove_Y;
		
	E_ManualJog.eMove_Y :;
		IF fbModuleAxis_Y.absPositionDone THEN
			eManualJog := E_ManualJog.eMove_Y_Done;
		END_IF
		
	E_ManualJog.eMove_Y_Done	:;
		eManualJog := E_ManualJog.eIdle;
	END_CASE
ELSE
	eManualJog := E_ManualJog.eIdle;
END_IF
                    
END_ACTION

ACTION ACT_InitListOfOffset:
                      up_Z_Position := -10;
nestNumber := 10;

arListXYZ_Offset[0].X_AxisOffsetPosition := 0;
arListXYZ_Offset[0].Y_AxisOffsetPosition := 0;
arListXYZ_Offset[0].Z_AxisOffsetPosition := 0;

arListXYZ_Offset[1].X_AxisOffsetPosition := 0;
arListXYZ_Offset[1].Y_AxisOffsetPosition := 0;
arListXYZ_Offset[1].Z_AxisOffsetPosition := -145;

arListXYZ_Offset[2].X_AxisOffsetPosition := 0;
arListXYZ_Offset[2].Y_AxisOffsetPosition := 40;
arListXYZ_Offset[2].Z_AxisOffsetPosition := -145;

arListXYZ_Offset[3].X_AxisOffsetPosition := 0;
arListXYZ_Offset[3].Y_AxisOffsetPosition := 80;
arListXYZ_Offset[3].Z_AxisOffsetPosition := -145;

arListXYZ_Offset[4].X_AxisOffsetPosition := 0;
arListXYZ_Offset[4].Y_AxisOffsetPosition := 120;
arListXYZ_Offset[4].Z_AxisOffsetPosition := -145;

arListXYZ_Offset[5].X_AxisOffsetPosition := 0;
arListXYZ_Offset[5].Y_AxisOffsetPosition := 160;
arListXYZ_Offset[5].Z_AxisOffsetPosition := -145;

arListXYZ_Offset[6].X_AxisOffsetPosition := 80;
arListXYZ_Offset[6].Y_AxisOffsetPosition := 80;
arListXYZ_Offset[6].Z_AxisOffsetPosition := -145;

arListXYZ_Offset[7].X_AxisOffsetPosition := 80;
arListXYZ_Offset[7].Y_AxisOffsetPosition := 40;
arListXYZ_Offset[7].Z_AxisOffsetPosition := -145;

arListXYZ_Offset[8].X_AxisOffsetPosition := 80;
arListXYZ_Offset[8].Y_AxisOffsetPosition := 80;
arListXYZ_Offset[8].Z_AxisOffsetPosition := -145;

arListXYZ_Offset[9].X_AxisOffsetPosition := 80;
arListXYZ_Offset[9].Y_AxisOffsetPosition := 120;
arListXYZ_Offset[9].Z_AxisOffsetPosition := -145;

arListXYZ_Offset[10].X_AxisOffsetPosition := 80;
arListXYZ_Offset[10].Y_AxisOffsetPosition := 160;
arListXYZ_Offset[10].Z_AxisOffsetPosition := -145;
                    
END_ACTION
END_PROGRAM

FUNCTION_BLOCK FB_BoxModeInterface
  VAR_IN_OUT
    virtualButtonAndSignal : UA_HMIVirtualButtonsAndSignals;
    Command_UnitMode : DINT;
    Command_UnnitModeChangeRequest : BOOL;
    Status_StateCurrent : DINT;
  END_VAR
  VAR
    modeState : E_PackModes := E_PackModes.Invalid;
    modeStringState : STRING := 'Invalid Mode';
    statecurrent : E_PackState;
  END_VAR

                  statecurrent := Status_StateCurrent;
Command_UnnitModeChangeRequest := TRUE;	// UnitModeChangeRequest can be managed depending on defined conditions (the user can modify them). It will allow a mode change if TRUE.


(*
 	Case to define what value will UnitCmd take depending on buttonState state.
*)
CASE statecurrent OF 
		
	E_PackState.eAborted : 
		IF virtualButtonAndSignal.In_VirtualManual THEN
			modeState := E_PackModes.Manual;
			modeStringState := 'Manual';
		ELSIF virtualButtonAndSignal.In_VirtualAuto THEN
			modeState := E_PackModes.Production;
			modeStringState := 'Production';
		END_IF

	E_PackState.eStopped :
		IF virtualButtonAndSignal.In_VirtualManual THEN
			modeState := E_PackModes.Manual;
			modeStringState := 'Manual';
		ELSIF virtualButtonAndSignal.In_VirtualAuto THEN
			modeState := E_PackModes.Production;
			modeStringState := 'Production';
		END_IF
		
	// More Unit modes can be defined. (look at E_PackModes)	

END_CASE

IF Command_UnnitModeChangeRequest THEN
	Command_UnitMode := modeState;
END_IF

                
END_FUNCTION_BLOCK

FUNCTION_BLOCK FB_BoxStateInterface
  VAR_IN_OUT
    realButtonAndSignal : UA_ButtonAndSignal;
    virtualButtonAndSignal : UA_HMIVirtualButtonsAndSignals;
    Command_CntrlCmd : DINT;
    Command_CmdChangeRequest : BOOL;
    Status_StateCurrent : DINT;
  END_VAR
  VAR
    cmdState : E_PackCmd := E_PackCmd.eUndefined;
    cmdStringState : STRING := 'Command undefined';
    memoryHold : BOOL;
    stateCurrent : E_PackState;
  END_VAR

                  stateCurrent := Status_StateCurrent;

(*
 	Case to define what value will CntrlCmd take depending on the Status_StateCurrent.
 	Depending on the current state, only certain commands will be allowed.
*)
CASE stateCurrent OF 
	
	E_PackState.eAborting :;	// no command can happen while aborting
	
	E_PackState.eAborted :
		IF realButtonAndSignal.In_Reset OR virtualButtonAndSignal.In_VirtualReset THEN //The Clearing will happen on a Reset so the Clear command is unused. Look at ISA-TR88.00.02-2022(It is common 
																					  // practice for Clear and Reset to be initiated using the same physical operator interface device)
			cmdState := E_PackCmd.eClear;
			cmdStringState := 'Clear';
		END_IF
		
	E_PackState.eClearing :
		IF NOT realButtonAndSignal.In_Estop OR virtualButtonAndSignal.In_VirtualAbort THEN
			cmdState := E_PackCmd.eAbort;
			cmdStringState := 'Abort';
		END_IF
	
	E_PackState.eStopped :
		IF NOT realButtonAndSignal.In_Estop OR virtualButtonAndSignal.In_VirtualAbort THEN
			cmdState := E_PackCmd.eAbort;
			cmdStringState := 'Abort';
		ELSIF realButtonAndSignal.In_Reset OR virtualButtonAndSignal.In_VirtualReset THEN
			cmdState := E_PackCmd.eReset;
			cmdStringState := 'Reset';
		END_IF
		
	E_PackState.eStopping :
		IF NOT realButtonAndSignal.In_Estop OR virtualButtonAndSignal.In_VirtualAbort THEN
			cmdState := E_PackCmd.eAbort;
			cmdStringState := 'Abort';
		END_IF
			
	E_PackState.eResetting : 
		IF NOT realButtonAndSignal.In_Estop OR virtualButtonAndSignal.In_VirtualAbort THEN
			cmdState := E_PackCmd.eAbort;
			cmdStringState := 'Abort';
		ELSIF realButtonAndSignal.In_Stop OR virtualButtonAndSignal.In_VirtualStop THEN
			cmdState := E_PackCmd.eStop;
			cmdStringState := 'Stop';
		END_IF
			
	E_PackState.eIdle :
		IF NOT realButtonAndSignal.In_Estop OR virtualButtonAndSignal.In_VirtualAbort THEN
			cmdState := E_PackCmd.eAbort;
			cmdStringState := 'Abort';
		ELSIF realButtonAndSignal.In_Stop OR virtualButtonAndSignal.In_VirtualStop THEN
			cmdState := E_PackCmd.eStop;
			cmdStringState := 'Stop';
		ELSIF realButtonAndSignal.In_Start OR virtualButtonAndSignal.In_VirtualStart THEN
			cmdState := E_PackCmd.eStart;
			cmdStringState := 'Start';
		END_IF
	
	E_PackState.eStarting :
		IF NOT realButtonAndSignal.In_Estop OR virtualButtonAndSignal.In_VirtualAbort THEN
			cmdState := E_PackCmd.eAbort;
			cmdStringState := 'Abort';
		ELSIF realButtonAndSignal.In_Stop OR virtualButtonAndSignal.In_VirtualStop THEN
			cmdState := E_PackCmd.eStop;
			cmdStringState := 'Stop';
		END_IF
		
	E_PackState.eExecute :
		IF NOT realButtonAndSignal.In_Estop OR virtualButtonAndSignal.In_VirtualAbort THEN
			cmdState := E_PackCmd.eAbort;
			cmdStringState := 'Abort';
		ELSIF realButtonAndSignal.In_Stop OR virtualButtonAndSignal.In_VirtualStop THEN
			cmdState := E_PackCmd.eStop;
			cmdStringState := 'Stop';
		ELSIF virtualButtonAndSignal.In_VirtualHold THEN
			cmdState := E_PackCmd.eHold;
			cmdStringState := 'Hold';
			memoryHold	:= TRUE;
		ELSIF (NOT GVL_Abox.uaAboxInterface.uaDigitalIn.Input_0_4) AND (NOT GVL_Abox.uaAboxInterface.uaDigitalIn.Input_0_5) AND (NOT GVL_Abox.uaAboxInterface.uaDigitalIn.Input_0_6) THEN // These buttons and sensors are only used as exemple to test.
			cmdState := E_PackCmd.eSuspend;
			cmdStringState := 'Suspend';
		ELSIF GVL_Abox.uaAboxInterface.uaDigitalIn.Input_0_1 THEN // These buttons and sensors are only used as exemple to test.
			cmdState := E_PackCmd.eComplete;
			cmdStringState := 'Complete';
		END_IF 
			
	E_PackState.eHolding :
		IF NOT realButtonAndSignal.In_Estop OR virtualButtonAndSignal.In_VirtualAbort THEN
			cmdState := E_PackCmd.eAbort;
			cmdStringState := 'Abort';
		ELSIF realButtonAndSignal.In_Stop OR virtualButtonAndSignal.In_VirtualStop THEN
			cmdState := E_PackCmd.eStop;
			cmdStringState := 'Stop';
		END_IF 
		
	E_PackState.eHeld :
		IF NOT realButtonAndSignal.In_Estop OR virtualButtonAndSignal.In_VirtualAbort THEN
			cmdState := E_PackCmd.eAbort;
			cmdStringState := 'Abort';
		ELSIF realButtonAndSignal.In_Stop OR virtualButtonAndSignal.In_VirtualStop THEN
			cmdState := E_PackCmd.eStop;
			cmdStringState := 'Stop';
		ELSIF memoryHold AND NOT virtualButtonAndSignal.In_VirtualHold THEN
			cmdState := E_PackCmd.eUnhold;
			cmdStringState	:= 'Unhold';
		END_IF 

	E_PackState.eUnholding :
		IF NOT realButtonAndSignal.In_Estop OR virtualButtonAndSignal.In_VirtualAbort THEN
			cmdState := E_PackCmd.eAbort;
			cmdStringState := 'Abort';
		ELSIF realButtonAndSignal.In_Stop OR virtualButtonAndSignal.In_VirtualStop THEN
			cmdState := E_PackCmd.eStop;
			cmdStringState := 'Stop';
		END_IF 
	
	E_PackState.eSuspending :
		IF NOT realButtonAndSignal.In_Estop OR virtualButtonAndSignal.In_VirtualAbort THEN
			cmdState := E_PackCmd.eAbort;
			cmdStringState := 'Abort';
		ELSIF realButtonAndSignal.In_Stop OR virtualButtonAndSignal.In_VirtualStop THEN
			cmdState := E_PackCmd.eStop;
			cmdStringState := 'Stop';
		END_IF 
			
	E_PackState.eSuspended :
		IF NOT realButtonAndSignal.In_Estop OR virtualButtonAndSignal.In_VirtualAbort THEN
			cmdState := E_PackCmd.eAbort;
			cmdStringState := 'Abort';
		ELSIF realButtonAndSignal.In_Stop OR virtualButtonAndSignal.In_VirtualStop THEN
			cmdState := E_PackCmd.eStop;
			cmdStringState := 'Stop';
		ELSIF GVL_Abox.uaAboxInterface.uaDigitalIn.Input_0_0 THEN // These buttons and sensors are only used as exemple to test.
			cmdState := E_PackCmd.eUnsuspend;
			cmdStringState := 'Unsuspend';
		END_IF 
		
	E_PackState.eUnsuspending :
		IF NOT realButtonAndSignal.In_Estop OR virtualButtonAndSignal.In_VirtualAbort THEN
			cmdState := E_PackCmd.eAbort;
			cmdStringState := 'Abort';
		ELSIF realButtonAndSignal.In_Stop OR virtualButtonAndSignal.In_VirtualStop THEN
			cmdState := E_PackCmd.eStop;
			cmdStringState := 'Stop';
		END_IF 
		
	E_PackState.eCompleting :
		IF NOT realButtonAndSignal.In_Estop OR virtualButtonAndSignal.In_VirtualAbort THEN
			cmdState := E_PackCmd.eAbort;
			cmdStringState := 'Abort';
		ELSIF realButtonAndSignal.In_Stop OR virtualButtonAndSignal.In_VirtualStop THEN
			cmdState := E_PackCmd.eStop;
			cmdStringState := 'Stop';
		END_IF 
			
	E_PackState.eCompleted :
		IF NOT realButtonAndSignal.In_Estop OR virtualButtonAndSignal.In_VirtualAbort THEN
			cmdState := E_PackCmd.eAbort;
			cmdStringState := 'Abort';
		ELSIF realButtonAndSignal.In_Stop OR virtualButtonAndSignal.In_VirtualStop THEN
			cmdState := E_PackCmd.eStop;
			cmdStringState := 'Stop';
		ELSIF realButtonAndSignal.In_Reset OR virtualButtonAndSignal.In_VirtualReset THEN
			cmdState := E_PackCmd.eReset;
			cmdStringState := 'Reset';
		END_IF 

END_CASE

Command_CmdChangeRequest := GVL_Abox.uaAboxInterface.uaDigitalIn.Input_1_0;	 // definition of CommandChangeRequest. If TRUE, will allow a state change to happen ( multiple conditions can be chosen for it to be TRUE, and not all states requires it TRUE to change.)
Command_CntrlCmd := cmdState;

                
END_FUNCTION_BLOCK

FUNCTION_BLOCK FB_BoxStopReasonID
  VAR_IN_OUT
    Admin_StopReasonId : DINT;
    Command_CntrlCmd : DINT;
    realButtonAndSignal : UA_ButtonAndSignal;
    virtualButtonAndSignal : UA_HMIVirtualButtonsAndSignals;
  END_VAR
  VAR
    StopReasonState : E_PackStopReasonId := E_PackStopReasonId.Undefined;
    StopReasonStringState : STRING := 'Undefined';
    cntrlCmd : E_PackCmd;
    globalButtonsAndSignals : UA_GlobalButtonsAndSignals;
  END_VAR

                  cntrlCmd := Command_CntrlCmd;
globalButtonsAndSignals.physicals := realButtonAndSignal;
globalButtonsAndSignals.virtuals := virtualButtonAndSignal;

(*
 	Case to define what value will StopReasonID take depending on cntrlCmd states.
*)
CASE cntrlCmd OF 
	
	E_PackCmd.eAbort :
		IF NOT globalButtonsAndSignals.physicals.In_Estop THEN
			StopReasonState := E_PackStopReasonId.RealEstopButtonPushed;
			StopReasonStringState := 'Physical EStop Button Pushed';
		ELSIF 
			globalButtonsAndSignals.virtuals.In_VirtualAbort THEN
			StopReasonState := E_PackStopReasonId.VirtualAbortButtonPushed;
			StopReasonStringState := 'Abort Screen Button Pushed';
		END_IF

	E_PackCmd.eStop :
		IF globalButtonsAndSignals.physicals.In_Stop THEN
			StopReasonState := E_PackStopReasonId.RealStopButtonPushed;
			StopReasonStringState := 'Physical Stop Button pushed';
		ELSIF globalButtonsAndSignals.virtuals.In_VirtualStop THEN
			StopReasonState := E_PackStopReasonId.VirtualStopButtonPushed;
			StopReasonStringState := 'Virtual Stop button pushed';
		END_IF
		
	E_PackCmd.eHold :	
		IF globalButtonsAndSignals.virtuals.In_VirtualHold THEN
			StopReasonState := E_PackStopReasonId.VirtualHoldButtonPushed;
			StopReasonStringState := 'Virtual Hold button pushed';
		END_IF
		
	// More StopReasonID can be defined. (look at E_PackStopReasonId)
	
	ELSE
        StopReasonState := E_PackStopReasonId.Undefined;
        StopReasonStringState := 'Undefined';
END_CASE

Admin_StopReasonId := StopReasonState;

                
END_FUNCTION_BLOCK

PROGRAM PRG_MapBox
  VAR
    SoftInOut_Command_UnitModeChangeRequest : BOOL;  (* ////////////////////////////////////////////////////// Soft In Out signals (Mainly for TP700 UI and Pack) ////////////////////////////////////////////////////// *)
    SoftInOut_Command_CmdChangeRequest : BOOL;
    SoftIn_PlcCycleTime : BYTE;  (* Used to check if read is running *)
    SoftIn_HmiControlsPbManual : BOOL;  (* See in HW for commande push buttons Linked to GVL_Abox...uaHmiVirtualButtonAndSignal *)
    SoftIn_HmiControlsPbAuto : BOOL;
    SoftIn_HmiControlsPbAbort : BOOL;
    SoftIn_HmiControlsPbStop : BOOL;
    SoftIn_HmiControlsPbReset : BOOL;
    SoftIn_HmiControlsPbStart : BOOL;
    SoftIn_HmiControlsPbHold : BOOL;
    SoftOut_PlcCycleTime : BYTE;  (* ////////////////////////////////////////////////////// Soft Out signals (Mainly for TP700 UI and Pack) ////////////////////////////////////////////////////// *)
    SoftOut_Idle : BOOL;  (* Linked to GVL_Abox...uaButtonAndSignal *)
    SoftOut_Execute : BOOL;
    SoftOut_Stopped : BOOL;
    SoftOut_Held : BOOL;
    SoftOut_Suspended : BOOL;
    SoftOut_packtag_admin_union_stopreasonid : HEVS_Min_PackTag_Union_Dint_FourBytesArray;  (* These six (6) variables are sent to Simatic then TP700 Linked to GVL_Abox..uaPackBox *)
    SoftOut_packtag_admin_union_curdisabledstates : HEVS_Min_PackTag_Union_Dword_Dint_FourBytesArray;
    SoftOut_packtag_status_union_unitmodecurrent : HEVS_Min_PackTag_Union_Dint_FourBytesArray;
    SoftOut_packtag_status_union_statecurrent : HEVS_Min_PackTag_Union_Dint_FourBytesArray;
    SoftOut_packtag_command_union_unitmode : HEVS_Min_PackTag_Union_Dint_FourBytesArray;
    SoftOut_packtag_command_union_cntrlcmd : HEVS_Min_PackTag_Union_Dint_FourBytesArray;
    HardIn_E_Stop : BOOL;  (* ////////////////////////////////////////////////////// Hardware In Out signal, (mainly linked to GVL_Abox GVL_Abox contains a Structure of Hardware Please link to GVL_Abox and not directly to Profinet ////////////////////////////////////////////////////// *)
    HardIn_ButtonReset : BOOL;
    HardIn_ButtonStart : BOOL;
    HardIn_ButtonStop : BOOL;
    HardIn_IOLink_port7_Balluf_Data1 : REAL;
    HardIn_IOLink_port7_Balluf_Data2 : REAL;
    HardIn_IOLink_port7_Balluf_Data3 : REAL;
    HardIn_IOLINK_Port7_ContactTemp_FourBytes : REAL;
    HardIn_IOLINK_Port7_Status_FourBytes : DWORD;
    HardIn_IOLINK_Port1_O300DL_Value : WORD;
    HardIn_IOLINK_Port1_O300DL_BCD1 : BOOL;
    HardIn_IOLINK_Port1_O300DL_Q : BOOL;
    HardIn_IOLINK_Port1_O300DL_A : BOOL;
    HardIn_IOLINK_Port2_O300ZL_BCD1 : BOOL;
    HardIn_IOLINK_Port2_O300ZL_Q : BOOL;
    HardIn_IOLINK_Port2_O300ZL_A : BOOL;
    HardIn_IOLINK_Port3_U300D50_Value : DWORD;
    HardIn_IOLINK_Port3_U300D50_Scale : SINT;
    HardIn_IOLINK_Port3_U300D50_SSC1 : BOOL;
    HardIn_IOLINK_Port3_U300D50_SSC2 : BOOL;
    HardIn_IOLINK_Port3_U300D50_Quality : BOOL;
    HardIn_IOLINK_Port3_U300D50_Alarm : BOOL;
    HardIn_IOLINK_Port3_U300D50_SSC4 : BOOL;
    HardIn_IOLINK_Port4_U300P50_Value : DWORD;
    HardIn_IOLINK_Port4_U300P50_Scale : SINT;
    HardIn_IOLINK_Port4_U300P50_SSC1 : BOOL;
    HardIn_IOLINK_Port4_U300P50_SSC2 : BOOL;
    HardIn_IOLINK_Port4_U300P50_Quality : BOOL;
    HardIn_IOLINK_Port4_U300P50_Alarm : BOOL;
    HardIn_IOLINK_Port4_U300P50_SSC4 : BOOL;
    HardIn_IOLINK_Port5_SchunkMMS22_Value : WORD;
    HardIn_BackPlane_DI_32_Input_0_0 : BOOL;
    HardIn_BackPlane_DI_32_Input_0_1 : BOOL;
    HardIn_BackPlane_DI_32_Input_0_2 : BOOL;
    HardIn_BackPlane_DI_32_Input_0_3 : BOOL;
    HardIn_BackPlane_DI_32_Input_0_4 : BOOL;
    HardIn_BackPlane_DI_32_Input_0_5 : BOOL;
    HardIn_BackPlane_DI_32_Input_0_6 : BOOL;
    HardIn_BackPlane_DI_32_Input_0_7 : BOOL;
    HardIn_BackPlane_DI_32_Input_1_0 : BOOL;
    HardIn_BackPlane_DI_32_Input_1_1 : BOOL;
    HardIn_BackPlane_DI_32_Input_1_2 : BOOL;
    HardIn_BackPlane_DI_32_Input_1_3 : BOOL;
    HardIn_BackPlane_DI_32_Input_1_4 : BOOL;
    HardIn_BackPlane_DI_32_Input_1_5 : BOOL;
    HardIn_BackPlane_DI_32_Input_1_6 : BOOL;
    HardIn_BackPlane_DI_32_Input_1_7 : BOOL;
    HardIn_BackPlane_DI_32_Input_2_0 : BOOL;
    HardIn_BackPlane_DI_32_Input_2_1 : BOOL;
    HardIn_BackPlane_DI_32_Input_2_2 : BOOL;
    HardIn_BackPlane_DI_32_Input_2_3 : BOOL;
    HardIn_BackPlane_DI_32_Input_2_4 : BOOL;
    HardIn_BackPlane_DI_32_Input_2_5 : BOOL;
    HardIn_BackPlane_DI_32_Input_2_6 : BOOL;
    HardIn_BackPlane_DI_32_Input_2_7 : BOOL;
    HardIn_BackPlane_DI_32_Input_3_0 : BOOL;
    HardIn_BackPlane_DI_32_Input_3_1 : BOOL;
    HardIn_BackPlane_DI_32_Input_3_2 : BOOL;
    HardIn_BackPlane_DI_32_Input_3_3 : BOOL;
    HardIn_BackPlane_DI_32_Input_3_4 : BOOL;
    HardIn_BackPlane_DI_32_Input_3_5 : BOOL;
    HardIn_BackPlane_DI_32_Input_3_6 : BOOL;
    HardIn_BackPlane_DI_32_Input_3_7 : BOOL;
    IOBackPlane_AnalogInput_IW4 : WORD;
    IOBackPlane_AnalogInput_IW6 : WORD;
    IOBackPlane_AnalogInput_IW8 : WORD;
    IOBackPlane_AnalogInput_IW10 : WORD;
    IOBackPlane_AnalogInput_IW12 : WORD;
    IOBackPlane_AnalogInput_IW14 : WORD;
    IOBackPlane_AnalogInput_IW16 : WORD;
    IOBackPlane_AnalogInput_IW18 : WORD;
    HardOut_IOLink_Port6_Festo_Valve : BOOL;
    HardOut_BackPlane_DO_32_output_0_0 : BOOL;  (* Digital Out *)
    HardOut_BackPlane_DO_32_output_0_1 : BOOL;
    HardOut_BackPlane_DO_32_output_0_2 : BOOL;
    HardOut_BackPlane_DO_32_output_0_3 : BOOL;
    HardOut_BackPlane_DO_32_output_0_4 : BOOL;
    HardOut_BackPlane_DO_32_output_0_5 : BOOL;
    HardOut_BackPlane_DO_32_output_0_6 : BOOL;
    HardOut_BackPlane_DO_32_output_0_7 : BOOL;
    HardOut_BackPlane_DO_32_output_1_0 : BOOL;
    HardOut_BackPlane_DO_32_output_1_1 : BOOL;
    HardOut_BackPlane_DO_32_output_1_2 : BOOL;
    HardOut_BackPlane_DO_32_output_1_3 : BOOL;
    HardOut_BackPlane_DO_32_output_1_4 : BOOL;
    HardOut_BackPlane_DO_32_output_1_5 : BOOL;
    HardOut_BackPlane_DO_32_output_1_6 : BOOL;
    HardOut_BackPlane_DO_32_output_1_7 : BOOL;
    HardOut_BackPlane_DO_32_output_2_0 : BOOL;
    HardOut_BackPlane_DO_32_output_2_1 : BOOL;
    HardOut_BackPlane_DO_32_output_2_2 : BOOL;
    HardOut_BackPlane_DO_32_output_2_3 : BOOL;
    HardOut_BackPlane_DO_32_output_2_4 : BOOL;
    HardOut_BackPlane_DO_32_output_2_5 : BOOL;
    HardOut_BackPlane_DO_32_output_2_6 : BOOL;
    HardOut_BackPlane_DO_32_output_2_7 : BOOL;
    HardOut_BackPlane_DO_32_output_3_0 : BOOL;
    HardOut_BackPlane_DO_32_output_3_1 : BOOL;
    HardOut_BackPlane_DO_32_output_3_2 : BOOL;
    HardOut_BackPlane_DO_32_output_3_3 : BOOL;
    HardOut_BackPlane_DO_32_output_3_4 : BOOL;
    HardOut_BackPlane_DO_32_output_3_5 : BOOL;
    HardOut_BackPlane_DO_32_output_3_6 : BOOL;
    HardOut_BackPlane_DO_32_output_3_7 : BOOL;
    HardOut_BackPlane_AO_QW4 : WORD;  (* Analog Out *)
    HardOut_BackPlane_AO_QW6 : WORD;
    HardOut_BackPlane_AO_QW8 : WORD;
    HardOut_BackPlane_AO_QW10 : WORD;
    HardIn_port7_Data1_FourBytes : ARRAY[1..4] OF BYTE;  (* Intermediate variables to manage WORD, DWORD and REAL values Used to manage Profinet bytes attribution *)
    HardIn_port7_Data2_FourBytes : ARRAY[1..4] OF BYTE;
    HardIn_port7_Data3_FourBytes : ARRAY[1..4] OF BYTE;
    HardIn_port7_ContTemp_FourBytes : ARRAY[1..4] OF BYTE;
    HardIn_port7_Stat_FourBytes : ARRAY[1..4] OF BYTE;
    HardIn_port1_Value_TwoBytes : ARRAY[1..2] OF BYTE;
    HardIn_port3_Value_FourBytes : ARRAY[1..4] OF BYTE;
    HardIn_port3_Scale_Byte : BYTE;
    HardIn_port4_Value_FourBytes : ARRAY[1..4] OF BYTE;
    HardIn_port4_Scale_Byte : BYTE;
    HardIn_port5_Value_TwoBytes : ARRAY[1..2] OF BYTE;
    fourBytesDW1 : DWORD;
    fourBytesPtR1 : POINTER TO REAL;
    fourBytesTest : ARRAY[1..4] OF BYTE;
    fourBytesDW2 : DWORD;
    fourBytesPtR2 : POINTER TO REAL;
    fourBytesDW3 : DWORD;
    fourBytesPtR3 : POINTER TO REAL;
    fourBytesDW4 : DWORD;
    fourBytesPtR4 : POINTER TO REAL;
    HardIn_IW4_TwoBytes : ARRAY[1..2] OF BYTE;  (* Analog Input via Profinet *)
    HardIn_IW6_TwoBytes : ARRAY[1..2] OF BYTE;
    HardIn_IW8_TwoBytes : ARRAY[1..2] OF BYTE;
    HardIn_IW10_TwoBytes : ARRAY[1..2] OF BYTE;
    HardIn_IW12_TwoBytes : ARRAY[1..2] OF BYTE;
    HardIn_IW14_TwoBytes : ARRAY[1..2] OF BYTE;
    HardIn_IW16_TwoBytes : ARRAY[1..2] OF BYTE;
    HardIn_IW18_TwoBytes : ARRAY[1..2] OF BYTE;
    HardOut_QW4_TwoBytes : ARRAY[1..2] OF BYTE;  (* Analog Output via Profinet *)
    HardOut_QW6_TwoBytes : ARRAY[1..2] OF BYTE;
    HardOut_QW8_TwoBytes : ARRAY[1..2] OF BYTE;
    HardOut_QW10_TwoBytes : ARRAY[1..2] OF BYTE;
    SoftOut_UnitMode_FourBytes : ARRAY[1..4] OF BYTE;  (* Soft Output via Profinet *)
    SoftOut_CntrlCmd_FourBytes : ARRAY[1..4] OF BYTE;
    SoftOut_stopReasonID_FourBytes : ARRAY[1..4] OF BYTE;
    SoftOut_CurDisabledStates_FourBytes : ARRAY[1..4] OF BYTE;
    SoftOut_UnitModeCurrent_FourBytes : ARRAY[1..4] OF BYTE;
    SoftOut_StateCurrent_FourBytes : ARRAY[1..4] OF BYTE;
  END_VAR

                  ///////////////////////////////////////////////////////// 
/// All GVL_Abox Links are processed in this ACTion
/////////////////////////////////////////////////////////
ACT_GVL_Abox();

(*
	Values to Profinet Station
*)
SoftOut_PlcCycleTime := SoftOut_PlcCycleTime + 1;
	
// Set PackML Status, Admin and Command values
SoftOut_packtag_admin_union_stopreasonid.DintAccess	:= GVL_Abox.uaPackBox.uAdmin_union_stopreasonid.DintAccess;
SoftOut_stopReasonID_FourBytes[1] 		:= SoftOut_packtag_admin_union_stopreasonid.FourBytesArrayAccess[4];
SoftOut_stopReasonID_FourBytes[2]		:= SoftOut_packtag_admin_union_stopreasonid.FourBytesArrayAccess[3];
SoftOut_stopReasonID_FourBytes[3] 		:= SoftOut_packtag_admin_union_stopreasonid.FourBytesArrayAccess[2];
SoftOut_stopReasonID_FourBytes[4] 		:= SoftOut_packtag_admin_union_stopreasonid.FourBytesArrayAccess[1];
	
SoftOut_packtag_admin_union_curdisabledstates.DwordAccess := GVL_Abox.uaPackBox.uAdmin_union_curdisabledstates.DwordAccess;
SoftOut_CurDisabledStates_FourBytes[1] 	:= SoftOut_packtag_admin_union_curdisabledstates.FourBytesArrayAccess[4];
SoftOut_CurDisabledStates_FourBytes[2] 	:= SoftOut_packtag_admin_union_curdisabledstates.FourBytesArrayAccess[3];
SoftOut_CurDisabledStates_FourBytes[3] 	:= SoftOut_packtag_admin_union_curdisabledstates.FourBytesArrayAccess[2];
SoftOut_CurDisabledStates_FourBytes[4] 	:= SoftOut_packtag_admin_union_curdisabledstates.FourBytesArrayAccess[1];
	
SoftOut_packtag_status_union_unitmodecurrent.DintAccess := GVL_Abox.uaPackBox.uStatus_union_unitmodecurrent .DintAccess;
SoftOut_UnitModeCurrent_FourBytes[1] 	:= SoftOut_packtag_status_union_unitmodecurrent.FourBytesArrayAccess[4];
SoftOut_UnitModeCurrent_FourBytes[2] 	:= SoftOut_packtag_status_union_unitmodecurrent.FourBytesArrayAccess[3];
SoftOut_UnitModeCurrent_FourBytes[3] 	:= SoftOut_packtag_status_union_unitmodecurrent.FourBytesArrayAccess[2];
SoftOut_UnitModeCurrent_FourBytes[4] 	:= SoftOut_packtag_status_union_unitmodecurrent.FourBytesArrayAccess[1];
	
SoftOut_packtag_status_union_statecurrent.DintAccess := GVL_Abox.uaPackBox.uStatus_union_statecurrent.DintAccess;
SoftOut_StateCurrent_FourBytes[1] 		:= SoftOut_packtag_status_union_statecurrent.FourBytesArrayAccess[4];
SoftOut_StateCurrent_FourBytes[2] 		:= SoftOut_packtag_status_union_statecurrent.FourBytesArrayAccess[3];
SoftOut_StateCurrent_FourBytes[3] 		:= SoftOut_packtag_status_union_statecurrent.FourBytesArrayAccess[2];
SoftOut_StateCurrent_FourBytes[4] 		:= SoftOut_packtag_status_union_statecurrent.FourBytesArrayAccess[1];
	
SoftOut_packtag_command_union_unitmode.DintAccess := GVL_Abox.uaPackBox.uCommand_union_unitmode.DintAccess;
SoftOut_UnitMode_FourBytes[1] 			:= SoftOut_packtag_command_union_unitmode.FourBytesArrayAccess[4];
SoftOut_UnitMode_FourBytes[2] 			:= SoftOut_packtag_command_union_unitmode.FourBytesArrayAccess[3];
SoftOut_UnitMode_FourBytes[3] 			:= SoftOut_packtag_command_union_unitmode.FourBytesArrayAccess[2];
SoftOut_UnitMode_FourBytes[4] 			:= SoftOut_packtag_command_union_unitmode.FourBytesArrayAccess[1];
	
SoftOut_packtag_command_union_cntrlcmd.DintAccess := GVL_Abox.uaPackBox.uCommand_union_cntrlcmd.DintAccess ;
SoftOut_CntrlCmd_FourBytes[1] 			:= SoftOut_packtag_command_union_cntrlcmd.FourBytesArrayAccess[4];
SoftOut_CntrlCmd_FourBytes[2] 			:= SoftOut_packtag_command_union_cntrlcmd.FourBytesArrayAccess[3];
SoftOut_CntrlCmd_FourBytes[3] 			:= SoftOut_packtag_command_union_cntrlcmd.FourBytesArrayAccess[2];
SoftOut_CntrlCmd_FourBytes[4] 			:= SoftOut_packtag_command_union_cntrlcmd.FourBytesArrayAccess[1];
	
SoftInOut_Command_UnitModeChangeRequest := GVL_Abox.uaPackBox.Command_UnitModeChangeRequest;
SoftInOut_Command_CmdChangeRequest 		:= GVL_Abox.uaPackBox.Command_CmdChangeRequest;

                

ACTION ACT_GVL_Abox:
                      ///////////////////////////////////////////////////////// 
/// All GVL_Abox Links are processed in this ACTion
/////////////////////////////////////////////////////////
    (*
        Values from Profinet Station
    *)
	
	// Management of REAL and WORD values
	fourBytesDW1 := SHL(TO_DWORD(HardIn_port7_Data1_FourBytes[1]),24) OR SHL(TO_DWORD(HardIn_port7_Data1_FourBytes[2]),16) OR SHL(TO_DWORD(HardIn_port7_Data1_FourBytes[3]),8) OR (TO_DWORD(HardIn_port7_Data1_FourBytes[4]));
	fourBytesPtR1 := ADR(fourBytesDW1);
	HardIn_IOLink_port7_Balluf_Data1 := fourBytesPtR1^;
	
	fourBytesDW2 := SHL(TO_DWORD(HardIn_port7_Data2_FourBytes[1]),24) OR SHL(TO_DWORD(HardIn_port7_Data2_FourBytes[2]),16) OR SHL(TO_DWORD(HardIn_port7_Data2_FourBytes[3]),8) OR (TO_DWORD(HardIn_port7_Data2_FourBytes[4]));
	fourBytesPtR2 := ADR(fourBytesDW2);
	HardIn_IOLink_port7_Balluf_Data2 := fourBytesPtR2^;
	
	fourBytesDW3 := SHL(TO_DWORD(HardIn_port7_Data3_FourBytes[1]),24) OR SHL(TO_DWORD(HardIn_port7_Data3_FourBytes[2]),16) OR SHL(TO_DWORD(HardIn_port7_Data3_FourBytes[3]),8) OR (TO_DWORD(HardIn_port7_Data3_FourBytes[4]));
	fourBytesPtR3 := ADR(fourBytesDW3);
	HardIn_IOLink_port7_Balluf_Data3 := fourBytesPtR3^;
	
	fourBytesDW4 := SHL(TO_DWORD(HardIn_port7_ContTemp_FourBytes[1]),24) OR SHL(TO_DWORD(HardIn_port7_ContTemp_FourBytes[2]),16) OR SHL(TO_DWORD(HardIn_port7_ContTemp_FourBytes[3]),8) OR (TO_DWORD(HardIn_port7_ContTemp_FourBytes[4]));
	fourBytesPtR4 := ADR(fourBytesDW4);
	HardIn_IOLINK_Port7_ContactTemp_FourBytes := fourBytesPtR4^;
	
	HardIn_IOLINK_Port7_Status_FourBytes := SHL(TO_DWORD(HardIn_port7_Stat_FourBytes[1]),24) OR SHL(TO_DWORD(HardIn_port7_Stat_FourBytes[2]),16) OR SHL(TO_DWORD(HardIn_port7_Stat_FourBytes[3]),8) OR (TO_DWORD(HardIn_port7_Stat_FourBytes[4]));
	HardIn_IOLINK_Port1_O300DL_Value := SHL(TO_WORD(HardIn_port1_Value_TwoBytes[1]),8) OR TO_WORD((HardIn_port1_Value_TwoBytes[2]));
	HardIn_IOLINK_Port3_U300D50_Value := SHL(TO_DWORD(HardIn_port3_Value_FourBytes[1]),24) OR SHL(TO_DWORD(HardIn_port3_Value_FourBytes[2]),16) OR SHL(TO_DWORD(HardIn_port3_Value_FourBytes[3]),8) OR (TO_DWORD(HardIn_port3_Value_FourBytes[4]));
	HardIn_IOLINK_Port3_U300D50_Scale := TO_SINT(HardIn_port3_Scale_Byte);
	HardIn_IOLINK_Port4_U300P50_Value := SHL(TO_DWORD(HardIn_port4_Value_FourBytes[1]),24) OR SHL(TO_DWORD(HardIn_port4_Value_FourBytes[2]),16) OR SHL(TO_DWORD(HardIn_port4_Value_FourBytes[3]),8) OR (TO_DWORD(HardIn_port4_Value_FourBytes[4]));
	HardIn_IOLINK_Port4_U300P50_Scale := TO_SINT(HardIn_port4_Scale_Byte);
	HardIn_IOLINK_Port5_SchunkMMS22_Value := SHL(TO_WORD(HardIn_port5_Value_TwoBytes[1]),8) OR TO_WORD((HardIn_port5_Value_TwoBytes[2]));
	
	IOBackPlane_AnalogInput_IW4		:= SHL(TO_WORD(HardIn_IW4_TwoBytes[1]),8) OR TO_WORD((HardIn_IW4_TwoBytes[2]));
	IOBackPlane_AnalogInput_IW6		:= SHL(TO_WORD(HardIn_IW6_TwoBytes[1]),8) OR TO_WORD((HardIn_IW6_TwoBytes[2]));
	IOBackPlane_AnalogInput_IW8		:= SHL(TO_WORD(HardIn_IW8_TwoBytes[1]),8) OR TO_WORD((HardIn_IW8_TwoBytes[2]));
	IOBackPlane_AnalogInput_IW10	:= SHL(TO_WORD(HardIn_IW10_TwoBytes[1]),8) OR TO_WORD((HardIn_IW10_TwoBytes[2]));
	IOBackPlane_AnalogInput_IW12	:= SHL(TO_WORD(HardIn_IW12_TwoBytes[1]),8) OR TO_WORD((HardIn_IW12_TwoBytes[2]));
	IOBackPlane_AnalogInput_IW14	:= SHL(TO_WORD(HardIn_IW14_TwoBytes[1]),8) OR TO_WORD((HardIn_IW14_TwoBytes[2]));
	IOBackPlane_AnalogInput_IW16	:= SHL(TO_WORD(HardIn_IW16_TwoBytes[1]),8) OR TO_WORD((HardIn_IW16_TwoBytes[2]));
	IOBackPlane_AnalogInput_IW18	:= SHL(TO_WORD(HardIn_IW18_TwoBytes[1]),8) OR TO_WORD((HardIn_IW18_TwoBytes[2]));
	
	
    
    // Get Value from Profinet Station with UA Client Write
	GVL_Abox.uaAboxInterface.uaButtonAndSignal.In_Estop     := HardIn_E_Stop;
	GVL_Abox.uaAboxInterface.uaButtonAndSignal.In_Reset     := HardIn_ButtonReset;
	GVL_Abox.uaAboxInterface.uaButtonAndSignal.In_Start     := HardIn_ButtonStart;
	GVL_Abox.uaAboxInterface.uaButtonAndSignal.In_Stop      := HardIn_ButtonStop;
	
    // Values from Balluff accelerometer
    GVL_Abox.uaAboxInterface.uaAccelerometer.Data_1         := HardIn_IOLink_port7_Balluf_Data1;
    GVL_Abox.uaAboxInterface.uaAccelerometer.Data_2         := HardIn_IOLink_port7_Balluf_Data2;
    GVL_Abox.uaAboxInterface.uaAccelerometer.Data_3         := HardIn_IOLink_port7_Balluf_Data3;
    GVL_Abox.uaAboxInterface.uaAccelerometer.Status         := HardIn_IOLINK_Port7_Status_FourBytes;
    GVL_Abox.uaAboxInterface.uaAccelerometer.Temperature    := HardIn_IOLINK_Port7_ContactTemp_FourBytes;

    // Values from Baumer O300 DL
    GVL_Abox.uaAboxInterface.uaO300_DL_Optic.Value          := HardIn_IOLINK_Port1_O300DL_Value;                
    GVL_Abox.uaAboxInterface.uaO300_DL_Optic.A              := HardIn_IOLINK_Port1_O300DL_A;                
    GVL_Abox.uaAboxInterface.uaO300_DL_Optic.Q              := HardIn_IOLINK_Port1_O300DL_Q;                
    GVL_Abox.uaAboxInterface.uaO300_DL_Optic.BCD1           := HardIn_IOLINK_Port1_O300DL_BCD1;     

    // Values from Baumer O300 ZL                
    GVL_Abox.uaAboxInterface.uaO300_ZL_Optic.A              := HardIn_IOLINK_Port2_O300ZL_A;                
    GVL_Abox.uaAboxInterface.uaO300_ZL_Optic.Q              := HardIn_IOLINK_Port2_O300ZL_Q;                
    GVL_Abox.uaAboxInterface.uaO300_ZL_Optic.BCD1           := HardIn_IOLINK_Port2_O300ZL_BCD1;                 

    // Values from Baumer U300 D50
    GVL_Abox.uaAboxInterface.uaU300_D50_Sound.Value         := HardIn_IOLINK_Port3_U300D50_Value;  
    GVL_Abox.uaAboxInterface.uaU300_D50_Sound.A             := HardIn_IOLINK_Port3_U300D50_Alarm;  
    GVL_Abox.uaAboxInterface.uaU300_D50_Sound.Q             := HardIn_IOLINK_Port3_U300D50_Quality;  
    GVL_Abox.uaAboxInterface.uaU300_D50_Sound.Scale         := HardIn_IOLINK_Port3_U300D50_Scale;  
    GVL_Abox.uaAboxInterface.uaU300_D50_Sound.SSC1          := HardIn_IOLINK_Port3_U300D50_SSC1;  
    GVL_Abox.uaAboxInterface.uaU300_D50_Sound.SSC2          := HardIn_IOLINK_Port3_U300D50_SSC2;  
    GVL_Abox.uaAboxInterface.uaU300_D50_Sound.SSC4          := HardIn_IOLINK_Port3_U300D50_SSC4;  
	
    // Values from Baumer U300 P50
    GVL_Abox.uaAboxInterface.uaU300_P50_Sound.Value         := HardIn_IOLINK_Port4_U300P50_Value;  
    GVL_Abox.uaAboxInterface.uaU300_P50_Sound.A             := HardIn_IOLINK_Port4_U300P50_Alarm;  
    GVL_Abox.uaAboxInterface.uaU300_P50_Sound.Q             := HardIn_IOLINK_Port4_U300P50_Quality;  
    GVL_Abox.uaAboxInterface.uaU300_P50_Sound.Scale         := HardIn_IOLINK_Port4_U300P50_Scale;  
    GVL_Abox.uaAboxInterface.uaU300_P50_Sound.SSC1          := HardIn_IOLINK_Port4_U300P50_SSC1;  
    GVL_Abox.uaAboxInterface.uaU300_P50_Sound.SSC2          := HardIn_IOLINK_Port4_U300P50_SSC2;  
    GVL_Abox.uaAboxInterface.uaU300_P50_Sound.SSC4          := HardIn_IOLINK_Port4_U300P50_SSC4;  
    
    // Values from Gripper sensor
    GVL_Abox.uaAboxInterface.uaSchunk.Value                 := HardIn_IOLINK_Port5_SchunkMMS22_Value;  
	
    // Get 32 Digital Input
    GVL_Abox.uaAboxInterface.uaDigitalIn.Input_0_0          := HardIn_BackPlane_DI_32_Input_0_0;
    GVL_Abox.uaAboxInterface.uaDigitalIn.Input_0_1          := HardIn_BackPlane_DI_32_Input_0_1;
    GVL_Abox.uaAboxInterface.uaDigitalIn.Input_0_2          := HardIn_BackPlane_DI_32_Input_0_2;
    GVL_Abox.uaAboxInterface.uaDigitalIn.Input_0_3          := HardIn_BackPlane_DI_32_Input_0_3;
    GVL_Abox.uaAboxInterface.uaDigitalIn.Input_0_4          := HardIn_BackPlane_DI_32_Input_0_4;
    GVL_Abox.uaAboxInterface.uaDigitalIn.Input_0_5          := HardIn_BackPlane_DI_32_Input_0_5;
    GVL_Abox.uaAboxInterface.uaDigitalIn.Input_0_6          := HardIn_BackPlane_DI_32_Input_0_6;
    GVL_Abox.uaAboxInterface.uaDigitalIn.Input_0_7          := HardIn_BackPlane_DI_32_Input_0_7;
    GVL_Abox.uaAboxInterface.uaDigitalIn.Input_1_0          := HardIn_BackPlane_DI_32_Input_1_0;
    GVL_Abox.uaAboxInterface.uaDigitalIn.Input_1_1          := HardIn_BackPlane_DI_32_Input_1_1;
    GVL_Abox.uaAboxInterface.uaDigitalIn.Input_1_2          := HardIn_BackPlane_DI_32_Input_1_2;
    GVL_Abox.uaAboxInterface.uaDigitalIn.Input_1_3          := HardIn_BackPlane_DI_32_Input_1_3;
    GVL_Abox.uaAboxInterface.uaDigitalIn.Input_1_4          := HardIn_BackPlane_DI_32_Input_1_4;
    GVL_Abox.uaAboxInterface.uaDigitalIn.Input_1_5          := HardIn_BackPlane_DI_32_Input_1_5;
    GVL_Abox.uaAboxInterface.uaDigitalIn.Input_1_6          := HardIn_BackPlane_DI_32_Input_1_6;
    GVL_Abox.uaAboxInterface.uaDigitalIn.Input_1_7          := HardIn_BackPlane_DI_32_Input_1_7;
    GVL_Abox.uaAboxInterface.uaDigitalIn.Input_2_0          := HardIn_BackPlane_DI_32_Input_2_0;
    GVL_Abox.uaAboxInterface.uaDigitalIn.Input_2_1          := HardIn_BackPlane_DI_32_Input_2_1;
    GVL_Abox.uaAboxInterface.uaDigitalIn.Input_2_2          := HardIn_BackPlane_DI_32_Input_2_2;
    GVL_Abox.uaAboxInterface.uaDigitalIn.Input_2_3          := HardIn_BackPlane_DI_32_Input_2_3;
    GVL_Abox.uaAboxInterface.uaDigitalIn.Input_2_4          := HardIn_BackPlane_DI_32_Input_2_4;
    GVL_Abox.uaAboxInterface.uaDigitalIn.Input_2_5          := HardIn_BackPlane_DI_32_Input_2_5;
    GVL_Abox.uaAboxInterface.uaDigitalIn.Input_2_6          := HardIn_BackPlane_DI_32_Input_2_6;
    GVL_Abox.uaAboxInterface.uaDigitalIn.Input_2_7          := HardIn_BackPlane_DI_32_Input_2_7;
    GVL_Abox.uaAboxInterface.uaDigitalIn.Input_3_0          := HardIn_BackPlane_DI_32_Input_3_0;
    GVL_Abox.uaAboxInterface.uaDigitalIn.Input_3_1          := HardIn_BackPlane_DI_32_Input_3_1;
    GVL_Abox.uaAboxInterface.uaDigitalIn.Input_3_2          := HardIn_BackPlane_DI_32_Input_3_2;
    GVL_Abox.uaAboxInterface.uaDigitalIn.Input_3_3          := HardIn_BackPlane_DI_32_Input_3_3;
    GVL_Abox.uaAboxInterface.uaDigitalIn.Input_3_4          := HardIn_BackPlane_DI_32_Input_3_4;
    GVL_Abox.uaAboxInterface.uaDigitalIn.Input_3_5          := HardIn_BackPlane_DI_32_Input_3_5;
    GVL_Abox.uaAboxInterface.uaDigitalIn.Input_3_6          := HardIn_BackPlane_DI_32_Input_3_6;
    GVL_Abox.uaAboxInterface.uaDigitalIn.Input_3_7          := HardIn_BackPlane_DI_32_Input_3_7;
	
	// Get 8 Analog Input
	GVL_Abox.uaAboxInterface.uaAnalogIn.IW_04 := IOBackPlane_AnalogInput_IW4;
	GVL_Abox.uaAboxInterface.uaAnalogIn.IW_06 := IOBackPlane_AnalogInput_IW6;
	GVL_Abox.uaAboxInterface.uaAnalogIn.IW_08 := IOBackPlane_AnalogInput_IW8;
	GVL_Abox.uaAboxInterface.uaAnalogIn.IW_10 := IOBackPlane_AnalogInput_IW10;
	GVL_Abox.uaAboxInterface.uaAnalogIn.IW_12 := IOBackPlane_AnalogInput_IW12;
	GVL_Abox.uaAboxInterface.uaAnalogIn.IW_14 := IOBackPlane_AnalogInput_IW14;
	GVL_Abox.uaAboxInterface.uaAnalogIn.IW_16 := IOBackPlane_AnalogInput_IW16;
	GVL_Abox.uaAboxInterface.uaAnalogIn.IW_18 := IOBackPlane_AnalogInput_IW18;
	
	// Get TP700 HMI Virtual Buttons value
	GVL_Abox.uaAboxInterface.uaHmiVirtualButtonAndSignal.In_VirtualManual := SoftIn_HmiControlsPbManual;
	GVL_Abox.uaAboxInterface.uaHmiVirtualButtonAndSignal.In_VirtualAuto := SoftIn_HmiControlsPbAuto;
	GVL_Abox.uaAboxInterface.uaHmiVirtualButtonAndSignal.In_VirtualAbort := SoftIn_HmiControlsPbAbort;
	GVL_Abox.uaAboxInterface.uaHmiVirtualButtonAndSignal.In_VirtualStop := SoftIn_HmiControlsPbStop;
	GVL_Abox.uaAboxInterface.uaHmiVirtualButtonAndSignal.In_VirtualReset := SoftIn_HmiControlsPbReset;
	GVL_Abox.uaAboxInterface.uaHmiVirtualButtonAndSignal.In_VirtualStart := SoftIn_HmiControlsPbStart;
	GVL_Abox.uaAboxInterface.uaHmiVirtualButtonAndSignal.In_VirtualHold := SoftIn_HmiControlsPbHold;

    // Set ABox Hardware Visual Signals
	SoftOut_Idle		:= GVL_Abox.uaAboxInterface.uaButtonAndSignal.Out_Idle;
	SoftOut_Execute 	:= GVL_Abox.uaAboxInterface.uaButtonAndSignal.Out_Execute;
	SoftOut_Stopped		:= GVL_Abox.uaAboxInterface.uaButtonAndSignal.Out_Stopped;
    
    // Set Gripper value
    HardOut_IOLink_Port6_Festo_Valve := NOT GVL_Abox.uaAboxInterface.uaSchunkGripper.SetOut;
    
    // Set 32 digital outputs
    HardOut_BackPlane_DO_32_output_0_0 := GVL_Abox.uaAboxInterface.uaDigitalOut.Output_0_0;
    HardOut_BackPlane_DO_32_output_0_1 := GVL_Abox.uaAboxInterface.uaDigitalOut.Output_0_1;
    HardOut_BackPlane_DO_32_output_0_2 := GVL_Abox.uaAboxInterface.uaDigitalOut.Output_0_2;
    HardOut_BackPlane_DO_32_output_0_3 := GVL_Abox.uaAboxInterface.uaDigitalOut.Output_0_3;
    HardOut_BackPlane_DO_32_output_0_4 := GVL_Abox.uaAboxInterface.uaDigitalOut.Output_0_4;
    HardOut_BackPlane_DO_32_output_0_5 := GVL_Abox.uaAboxInterface.uaDigitalOut.Output_0_5;
    HardOut_BackPlane_DO_32_output_0_6 := GVL_Abox.uaAboxInterface.uaDigitalOut.Output_0_6;
    HardOut_BackPlane_DO_32_output_0_7 := GVL_Abox.uaAboxInterface.uaDigitalOut.Output_0_7;
	
    HardOut_BackPlane_DO_32_output_1_0 := GVL_Abox.uaAboxInterface.uaDigitalOut.Output_1_0;
    HardOut_BackPlane_DO_32_output_1_1 := GVL_Abox.uaAboxInterface.uaDigitalOut.Output_1_1;
    HardOut_BackPlane_DO_32_output_1_2 := GVL_Abox.uaAboxInterface.uaDigitalOut.Output_1_2;
    HardOut_BackPlane_DO_32_output_1_3 := GVL_Abox.uaAboxInterface.uaDigitalOut.Output_1_3;
    HardOut_BackPlane_DO_32_output_1_4 := GVL_Abox.uaAboxInterface.uaDigitalOut.Output_1_4;
    HardOut_BackPlane_DO_32_output_1_5 := GVL_Abox.uaAboxInterface.uaDigitalOut.Output_1_5;
    HardOut_BackPlane_DO_32_output_1_6 := GVL_Abox.uaAboxInterface.uaDigitalOut.Output_1_6;
    HardOut_BackPlane_DO_32_output_1_7 := GVL_Abox.uaAboxInterface.uaDigitalOut.Output_1_7;
	
    HardOut_BackPlane_DO_32_output_2_0 := GVL_Abox.uaAboxInterface.uaDigitalOut.Output_2_0;
    HardOut_BackPlane_DO_32_output_2_1 := GVL_Abox.uaAboxInterface.uaDigitalOut.Output_2_1;
    HardOut_BackPlane_DO_32_output_2_2 := GVL_Abox.uaAboxInterface.uaDigitalOut.Output_2_2;
    HardOut_BackPlane_DO_32_output_2_3 := GVL_Abox.uaAboxInterface.uaDigitalOut.Output_2_3;
    HardOut_BackPlane_DO_32_output_2_4 := GVL_Abox.uaAboxInterface.uaDigitalOut.Output_2_4;
    HardOut_BackPlane_DO_32_output_2_5 := GVL_Abox.uaAboxInterface.uaDigitalOut.Output_2_5;
    HardOut_BackPlane_DO_32_output_2_6 := GVL_Abox.uaAboxInterface.uaDigitalOut.Output_2_6;
    HardOut_BackPlane_DO_32_output_2_7 := GVL_Abox.uaAboxInterface.uaDigitalOut.Output_2_7;
	
    HardOut_BackPlane_DO_32_output_3_0 := GVL_Abox.uaAboxInterface.uaDigitalOut.Output_3_0;
    HardOut_BackPlane_DO_32_output_3_1 := GVL_Abox.uaAboxInterface.uaDigitalOut.Output_3_1;
    HardOut_BackPlane_DO_32_output_3_2 := GVL_Abox.uaAboxInterface.uaDigitalOut.Output_3_2;
    HardOut_BackPlane_DO_32_output_3_3 := GVL_Abox.uaAboxInterface.uaDigitalOut.Output_3_3;
    HardOut_BackPlane_DO_32_output_3_4 := GVL_Abox.uaAboxInterface.uaDigitalOut.Output_3_4;
    HardOut_BackPlane_DO_32_output_3_5 := GVL_Abox.uaAboxInterface.uaDigitalOut.Output_3_5;
    HardOut_BackPlane_DO_32_output_3_6 := GVL_Abox.uaAboxInterface.uaDigitalOut.Output_3_6;
    HardOut_BackPlane_DO_32_output_3_7 := GVL_Abox.uaAboxInterface.uaDigitalOut.Output_3_7;
	
	// Set 32 analog outputs
	HardOut_BackPlane_AO_QW4	:= GVL_Abox.uaAboxInterface.uaAnalogOut.QW_04;
	HardOut_QW4_TwoBytes[1] 	:= TO_BYTE(SHR(HardOut_BackPlane_AO_QW4,8));
	HardOut_QW4_TwoBytes[2] 	:= TO_BYTE(HardOut_BackPlane_AO_QW4 AND 255);
	
	HardOut_BackPlane_AO_QW6	:= GVL_Abox.uaAboxInterface.uaAnalogOut.QW_06;
	HardOut_QW6_TwoBytes[1] 	:= TO_BYTE(SHR(HardOut_BackPlane_AO_QW6,8));
	HardOut_QW6_TwoBytes[2] 	:= TO_BYTE(HardOut_BackPlane_AO_QW6 AND 255);
	
	HardOut_BackPlane_AO_QW8	:= GVL_Abox.uaAboxInterface.uaAnalogOut.QW_08;
	HardOut_QW8_TwoBytes[1] 	:= TO_BYTE(SHR(HardOut_BackPlane_AO_QW8,8));
	HardOut_QW8_TwoBytes[2] 	:= TO_BYTE(HardOut_BackPlane_AO_QW8 AND 255);
	
	HardOut_BackPlane_AO_QW10	:= GVL_Abox.uaAboxInterface.uaAnalogOut.QW_10;
	HardOut_QW10_TwoBytes[1] 	:= TO_BYTE(SHR(HardOut_BackPlane_AO_QW10,8));
	HardOut_QW10_TwoBytes[2] 	:= TO_BYTE(HardOut_BackPlane_AO_QW10 AND 255);

                    
END_ACTION
END_PROGRAM

PROGRAM PRG_DeviceManager
  VAR
    SetOpenGripper : BOOL;  (* Gripper Pneumatic Device *)
    SetCloseGripper : BOOL;
    GetGripperSensor_mm : REAL;  (* Gripper Sensor Device *)
    gripperSensor : WORD;
  END_VAR

                  (* Manage IO*)
gripperSensor := GVL_Abox.uaAboxInterface.uaSchunk.Value;

(*
	Gripper Pneumatic Device
*)
IF SetOpenGripper THEN
	// Reset value after receiving a message
	SetOpenGripper := FALSE;
	GVL_Abox.uaAboxInterface.uaSchunkGripper.SetOut := TRUE;
END_IF

IF SetCloseGripper THEN
	// Reset value after receiving a message
	SetCloseGripper := FALSE;
	GVL_Abox.uaAboxInterface.uaSchunkGripper.SetOut := FALSE;
END_IF

(*
	Gripper Sensor Device
*)
GetGripperSensor_mm := WORD_TO_REAL(gripperSensor) * 0.01;


                
END_PROGRAM

PROGRAM PRG_PackUpdate

                  PackTag.Status.Parameter_Lreal[1].ID := 1001;
PackTag.Status.Parameter_Lreal[1].Name := 'Axes Velocity';
PackTag.Status.Parameter_Lreal[1].Unit := 'm/s';
PackTag.Status.Parameter_Lreal[1].Value := PRG_Process.stSetParam.rVelocity_m_s;

PackTag.Status.Parameter_Lreal[2].ID := 1002;
PackTag.Status.Parameter_Lreal[2].Name := 'Axes Acceleration';
PackTag.Status.Parameter_Lreal[2].Unit := 'm/s2';
PackTag.Status.Parameter_Lreal[2].Value := PRG_Process.stSetParam.rAcceleration_m_s2;

PackTag.Status.Parameter_Lreal[3].ID := 1003;
PackTag.Status.Parameter_Lreal[3].Name := 'Axes Deceleration';
PackTag.Status.Parameter_Lreal[3].Unit := 'm/s2';
PackTag.Status.Parameter_Lreal[3].Value := PRG_Process.stSetParam.rDeceleration_m_s2;

PackTag.Status.Parameter_Lreal[4].ID := 1004;
PackTag.Status.Parameter_Lreal[4].Name := 'Axes Jerk';
PackTag.Status.Parameter_Lreal[4].Unit := 'm/s3';
PackTag.Status.Parameter_Lreal[4].Value := PRG_Process.stSetParam.rJerk_m_s3;

                
END_PROGRAM

PROGRAM PRG_PackModule_Template
  VAR_IN_OUT
    Status_StateCurrent : DINT;  (* has to take the PackTag Status.StateCurrent *)
  END_VAR
  VAR
    stateLastCycie : E_PackState := E_PackState.eUndefined;  (* Store last cycle at the en of FB call to detect and state change Used to force minimum of one testSC.In = 0 and reset SC once between each SC *)
    actualState : E_PackState := E_PackState.eAborted;
    uliLoop : ULINT;
    init : BOOL;
    testSC : TON;
    setSC : BOOL;  (* This Flag is used as result on SC State complete. *)
    stActing : ST_Acting;
    LockResetting : BOOL;  (* For test, wait variable TRUE for resetting SC *)
  END_VAR

                  IF NOT init THEN
    init := TRUE;
END_IF
actualState := Status_StateCurrent;

(*
	Your code here
	For code in States, modify the actions. ACT
	
	Code for mode is still not impletemented
*)

ACT_Aborting();
ACT_Clearing();
ACT_Completing();
ACT_Execute();
ACT_Holding();
ACT_Resetting();
ACT_Starting();
ACT_Stopping();
ACT_Suspending();
ACT_Unholding();
ACT_Unsuspending();

(*
	Footer, do not modify the code below.

	For test of State Machine, we use a timer.
	Its allow to have some time to visualise it
	We should remove this timer in production version
*)
testSC(IN := stActing.Clearing_SC 		OR
             stActing.Starting_SC      	OR
             stActing.Execute_SC       	OR
             stActing.Stopping_SC      	OR
             stActing.Aborting_SC      	OR
             stActing.Holding_SC       	OR
             stActing.Unholding_SC     	OR
             stActing.Suspending_SC		OR
             stActing.Unsuspending_SC	OR
             stActing.Resetting_SC     	OR
             stActing.Completing_SC,
        PT := T#500MS); 
           
// State Complete if setSC is TRUE,
setSC := testSC.Q AND (stateLastCycie = actualState);

// This Statement MUST be written AFTER evaluation of setSC
stateLastCycie := actualState;
                

ACTION ACT_Aborting:
                      (*
	Manage Aborting
*)
IF actualState = E_PackState.eAborting THEN
	// Set to TRUE if no action requested
	stActing.Aborting_SC := TRUE;
ELSE
	stActing.Aborting_SC := FALSE;
END_IF

                    
END_ACTION

ACTION ACT_Clearing:
                      (*
	Manage Clearing
*)
IF actualState = E_PackState.eClearing THEN
	// Set to TRUE if no action requested
	stActing.Clearing_SC := TRUE;
ELSE
	stActing.Clearing_SC := FALSE;
END_IF
                    
END_ACTION

ACTION ACT_Completing:
                      (*
	Manage Completing
*)
IF actualState = E_PackState.eCompleting THEN
	// Set to TRUE if no action requested
	stActing.Completing_SC := TRUE;
ELSE
	stActing.Completing_SC := FALSE;
END_IF

                    
END_ACTION

ACTION ACT_Execute:
                      
                    
END_ACTION

ACTION ACT_Holding:
                      (*
	Manage Holding
*)
IF actualState = E_PackState.eHolding THEN
	// Set to TRUE if no action requested
	stActing.Holding_SC := TRUE;
ELSE
	stActing.Holding_SC := FALSE;
END_IF
                    
END_ACTION

ACTION ACT_Resetting:
                      (*
	Manage Resetting
*)
IF actualState = E_PackState.eResetting THEN
	// Set to TRUE if no action requested
	IF NOT LockResetting THEN
		stActing.Resetting_SC := TRUE;
	ELSE
		stActing.Resetting_SC := FALSE;		
	END_IF

ELSE
	stActing.Resetting_SC := FALSE;
END_IF
                    
END_ACTION

ACTION ACT_Starting:
                      (*
	Manage Starting
*)
IF actualState = E_PackState.eStarting THEN
	// Set to TRUE if no action requested
	stActing.Starting_SC := TRUE;
ELSE
	stActing.Starting_SC := FALSE;
END_IF
                    
END_ACTION

ACTION ACT_Stopping:
                      (*
	Manage Stopping
*)
IF actualState = E_PackState.eStopping THEN
	// Set to TRUE if no action requested
	stActing.Stopping_SC := TRUE;
ELSE
	stActing.Stopping_SC := FALSE;
END_IF
                    
END_ACTION

ACTION ACT_Suspending:
                      (*
	Manage Suspending
*)
IF actualState = E_PackState.eSuspending THEN
	// Set to TRUE if no action requested
	stActing.Suspending_SC := TRUE;
ELSE
	stActing.Suspending_SC := FALSE;
END_IF
                    
END_ACTION

ACTION ACT_Unholding:
                      (*
	Manage Unholding
*)
IF actualState = E_PackState.eUnholding THEN
	// Set to TRUE if no action requested
	stActing.Unholding_SC := TRUE;
ELSE
	stActing.Unholding_SC := FALSE;
END_IF
                    
END_ACTION

ACTION ACT_Unsuspending:
                      (*
	Manage Unsuspending
*)
IF actualState = E_PackState.eUnsuspending THEN
	// Set to TRUE if no action requested
	stActing.Unsuspending_SC := TRUE;
ELSE
	stActing.Unsuspending_SC := FALSE;
END_IF
                    
END_ACTION

PROPERTY SC : BOOL
GET
                          SC := setSC;
                        
END_GET
END_PROPERTY
END_PROGRAM

PROGRAM PRG_Student

                  
                
END_PROGRAM

CONFIGURATION Application
  RESOURCE Application ON PLC
    {attribute 'qualified_only'}
    VAR_GLOBAL CONSTANT  (* HEVS_PackTag_GVL - List of PackTags based on ISA–TR88.00.02-2022 www.hevs.ch Institut Systemes Industriels / Power & Control Project: Automation Box CtrlX S3 Author: Romain Ferrari & Cedric Lenoir Date: 2024 July 31 !!!!!! The value of these constants have to be set by the user depending on the system it is implemented on. !!!!!!\\ *)
      C_MAXSTATES : INT := 17;  (* Max State number. 0 is invalid *)
      C_COMMAND_MAXREALPARAMS : INT := 8;
      C_COMMAND_MAXSTRINGPARAMS : INT := 2;  (* / *)
      C_COMMAND_MAXLREALPARAMS : INT := 8;  (* Used in one of the main PackTag branch of the HEVS_PackTag_V30 : Command *)
      C_COMMAND_MAXDINTPARAMS : INT := 8;
      C_COMMAND_MAXRECIPE : INT := 8;
      C_STATUS_MAXREALPARAMS : INT := 8;  (* / *)
      C_STATUS_MAXSTRINGPARAMS : INT := 2;  (* / *)
      C_STATUS_MAXLREALPARAMS : INT := 8;
      C_STATUS_MAXDINTPARAMS : INT := 8;  (* Used in one of the main PackTag branch of the HEVS_PackTag_V30 : Status *)
      C_STATUS_MAXRECIPE : INT := 8;
      C_STATUS_MAXSTACKLIGHT : INT := 8;
      C_ADMIN_MAXREALPARAMS : INT := 8;  (* / *)
      C_ADMIN_MAXSTRINGPARAMS : INT := 2;  (* / *)
      C_ADMIN_MAXLREALPARAMS : INT := 8;
      C_ADMIN_MAXDINTPARAMS : INT := 8;
      C_ADMIN_MAXALARMS : INT := 20;
      C_ADMIN_MAXHISTORYALARMS : INT := 20;
      C_ADMIN_MAXWARNINGS : INT := 20;
      C_ADMIN_MAXCUMULATIVETIMES : INT := 3;  (* Minimum is 0 for [0], Arbitrarily initialized to 3 *)
      C_ADMIN_MAXPRODUCTDATA : INT := 11;
      C_ADMIN_MAXDISABLEDSTATES : INT := 8;
      C_ADMIN_MAXMODESTRANSITION : INT := 8;  (* is absolutely limited by C_ADMIN_MAXMODESTRANSITIONPACK *)
      C_ADMIN_MAXMODESTRANSITIONPACK : INT := 31;  (* as Pack used DWORD and 0 is reserved, max is limited to 31 *)
      C_MAXMODSTATESTIMES : INT := 8;
      C_MAXREALVARIABLES : INT := 8;
      C_MAXSTRINGVARIABLES : INT := 8;
      C_MAXLREALVARIABLES : INT := 8;
      C_MAXDINTVARIABLES : INT := 8;  (* Used in lower branches of the HEVS_PackTag_V30 *)
      C_MAXREALINGREDIENTS : INT := 8;
      C_MAXSTRINGINGREDIENTS : INT := 8;
      C_MAXLREALINGREDIENTS : INT := 8;
      C_MAXDINTINGREDIENTS : INT := 8;
      hevs_min_packtag_v2022 : HEVS_Min_PackTag_V2022;
    END_VAR
    {attribute 'qualified_only'}
    VAR_GLOBAL  (* PackTag - www.hevs.ch Institut Systemes Industriels Project: HEVS Pack 2022 Author: Cedric Lenoir Date: 2024 August 29 Base GVL for HEVS Pack Tag File name should be PackTag *)
      Command : HEVS_PackTag_Command;
      Status : HEVS_PackTag_Status;
      Admin : HEVS_PackTag_Admin;
      hevsPackTime : HEVS_Time;  (* HEVS Time, needed for Alarms and Time in Pack Computed with PRG_GetTime_CtrlX or PRG_GetTime_TwinCAT or Your own system *)
      hevsUI : HEVS_PackTag_UI;  (* Help for interface and diagnostic HEVS Pack could be used without this Struct. Can be used with fbCmdBoolInterface Can be used with fbGetActualBoolState *)
      hevsPackAlarm_UI : HEVS_PackAlarm_UI;  (* Help for interface and diagnostic HEVS Pack could be used without this Struct. Can be used with program PRG_TestAlarm *)
    END_VAR
    {attribute 'qualified_only'}
    VAR_GLOBAL  (* GVL_Node - Some GVL to test var with NodeRED. Source: www.hevs.ch Author: Cedric Lenoir Date: 22 August 2024 *)
      readREAL : REAL;
      readDINT : DINT;
      readBOOL : BOOL;
      readString : STRING;
      writeREAL : REAL;
      writeDINT : DINT;
      writeBOOL : BOOL;
    END_VAR
    {attribute 'qualified_only'}
    VAR_GLOBAL  (* GVL_AxisDefines *)
      X_Axis : MB_AXISIF_REF := (AxisName := 'Axis_x', AxisNo := 1);
      Y_Axis : MB_AXISIF_REF := (AxisName := 'Axis_y', AxisNo := 2);
      Z_Axis : MB_AXISIF_REF := (AxisName := 'Axis_z', AxisNo := 3);
    END_VAR
    {attribute 'qualified_only'}
    VAR_GLOBAL  (* GVL_Abox *)
      uaAboxInterface : UA_AboxInterface;  (* Hardware commands (and soft buttons) *)
      uaPackBox : UA_PackBox;  (* See header of UA_PackBox for more info. *)
    END_VAR
    TASK MainTask(INTERVAL := T#40ms, PRIORITY := 30);
    PROGRAM PLC_PACK WITH MainTask : PLC_PACK;
    PROGRAM PRG_TestAlarm WITH MainTask : PRG_TestAlarm;
    PROGRAM PRG_Sandbox WITH MainTask : PRG_Sandbox;
    PROGRAM PRG_GetTime_CtrlX WITH MainTask : PRG_GetTime_CtrlX;
    PROGRAM PRG_MapBox WITH MainTask : PRG_MapBox;
    PROGRAM PRG_DeviceManager WITH MainTask : PRG_DeviceManager;
    PROGRAM PRG_Process WITH MainTask : PRG_Process;
  END_RESOURCE
END_CONFIGURATION
